Yaskawa INFORM job: A_ROOF_SIDE_0617_2_PAINT_28.JBI

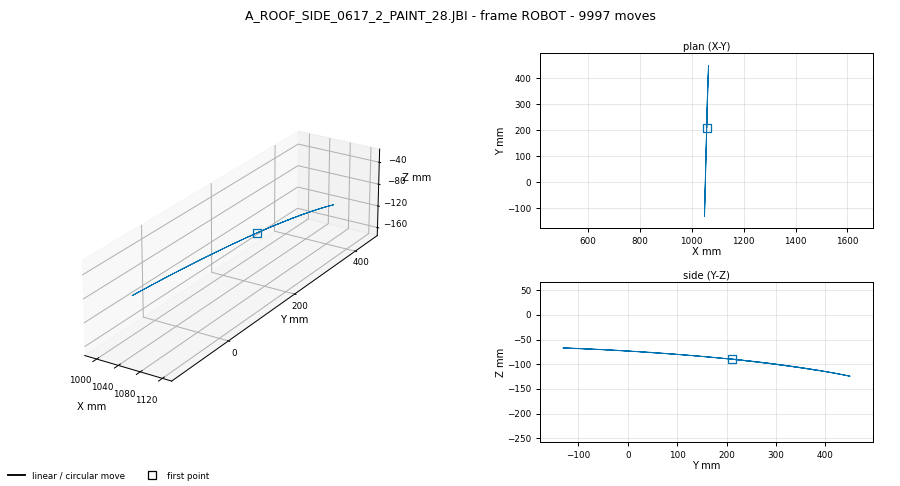
[picture p0: tool path of A_ROOF_SIDE_0617_2_PAINT_28.JBI in frame ROBOT, 9997 of 9997 moves have a stored position in this frame; points joined in program order, loops and branches not executed]
/JOB
//NAME A_ROOF_SIDE_0617_2_PAINT28
//POS
///NPOS 9997,0,0,0,0,0
///TOOL 1
///USER 0
///POSTYPE ROBOT
///RECTAN
///RCONF 1,0,0,0,0,0,0,0,0,0,0,0,0,0,0,0,0,0,0,0,0,0,0,0
C00000=1058.652,210.602,-89.176,172.510,33.165,156.166
C00001=1058.658,210.851,-89.202,172.512,33.168,156.167
C00002=1058.665,211.100,-89.228,172.514,33.173,156.168
C00003=1058.671,211.349,-89.254,172.516,33.176,156.168
C00004=1058.677,211.597,-89.280,172.518,33.181,156.169
C00005=1058.683,211.846,-89.306,172.520,33.184,156.170
C00006=1058.690,212.094,-89.332,172.522,33.189,156.171
C00007=1058.695,212.343,-89.358,172.524,33.192,156.171
C00008=1058.702,212.591,-89.384,172.526,33.196,156.172
C00009=1058.708,212.840,-89.410,172.528,33.200,156.173
C00010=1058.714,213.088,-89.436,172.530,33.204,156.174
C00011=1058.721,213.337,-89.461,172.531,33.208,156.174
C00012=1058.726,213.585,-89.488,172.533,33.212,156.175
C00013=1058.733,213.834,-89.513,172.535,33.216,156.176
C00014=1058.738,214.082,-89.540,172.537,33.220,156.177
C00015=1058.745,214.331,-89.565,172.539,33.224,156.177
C00016=1058.751,214.580,-89.592,172.541,33.227,156.178
C00017=1058.759,214.908,-89.627,172.544,33.233,156.179
C00018=1058.767,215.238,-89.662,172.546,33.238,156.180
C00019=1058.775,215.566,-89.696,172.549,33.243,156.181
C00020=1058.783,215.895,-89.731,172.553,33.248,156.182
C00021=1058.789,216.144,-89.756,172.555,33.253,156.183
C00022=1058.795,216.392,-89.783,172.557,33.256,156.184
C00023=1058.802,216.641,-89.810,172.559,33.260,156.184
C00024=1058.808,216.890,-89.835,172.561,33.264,156.185
C00025=1058.814,217.138,-89.862,172.563,33.268,156.186
C00026=1058.820,217.386,-89.888,172.565,33.271,156.186
C00027=1058.827,217.636,-89.914,172.567,33.276,156.187
C00028=1058.832,217.884,-89.941,172.569,33.279,156.188
C00029=1058.839,218.132,-89.967,172.571,33.284,156.189
C00030=1058.845,218.380,-89.993,172.573,33.287,156.189
C00031=1058.851,218.630,-90.019,172.575,33.291,156.190
C00032=1058.857,218.878,-90.046,172.577,33.295,156.191
C00033=1058.864,219.126,-90.072,172.579,33.299,156.192
C00034=1058.870,219.375,-90.099,172.581,33.302,156.192
C00035=1058.876,219.624,-90.125,172.583,33.307,156.193
C00036=1058.882,219.872,-90.151,172.585,33.310,156.194
C00037=1058.888,220.121,-90.177,172.587,33.314,156.194
C00038=1058.895,220.369,-90.204,172.589,33.318,156.195
C00039=1058.901,220.618,-90.230,172.591,33.322,156.196
C00040=1058.907,220.866,-90.256,172.593,33.326,156.197
C00041=1058.914,221.102,-90.282,172.595,33.329,156.197
C00042=1058.918,221.337,-90.307,172.598,33.333,156.198
C00043=1058.925,221.573,-90.333,172.600,33.337,156.199
C00044=1058.930,221.809,-90.357,172.601,33.340,156.199
C00045=1058.936,222.045,-90.382,172.603,33.344,156.200
C00046=1058.942,222.280,-90.407,172.605,33.348,156.201
C00047=1058.948,222.516,-90.433,172.607,33.351,156.202
C00048=1058.954,222.752,-90.458,172.609,33.355,156.202
C00049=1058.959,223.000,-90.485,172.611,33.359,156.203
C00050=1058.966,223.249,-90.512,172.613,33.363,156.204
C00051=1058.972,223.498,-90.538,172.615,33.367,156.205
C00052=1058.977,223.746,-90.565,172.617,33.371,156.205
C00053=1058.985,223.995,-90.591,172.619,33.374,156.206
C00054=1058.990,224.243,-90.618,172.621,33.379,156.207
C00055=1058.996,224.491,-90.645,172.623,33.382,156.207
C00056=1059.003,224.740,-90.672,172.626,33.386,156.208
C00057=1059.009,224.988,-90.699,172.628,33.390,156.209
C00058=1059.016,225.237,-90.725,172.630,33.394,156.210
C00059=1059.021,225.485,-90.752,172.632,33.397,156.210
C00060=1059.027,225.734,-90.779,172.635,33.402,156.211
C00061=1059.034,225.983,-90.806,172.637,33.405,156.212
C00062=1059.039,226.231,-90.832,172.639,33.409,156.212
C00063=1059.045,226.479,-90.859,172.641,33.413,156.213
C00064=1059.053,226.728,-90.886,172.643,33.417,156.214
C00065=1059.058,226.976,-90.913,172.645,33.421,156.215
C00066=1059.065,227.225,-90.940,172.647,33.424,156.215
C00067=1059.070,227.473,-90.966,172.649,33.428,156.216
C00068=1059.077,227.722,-90.993,172.651,33.432,156.217
C00069=1059.083,227.970,-91.021,172.654,33.436,156.218
C00070=1059.090,228.219,-91.047,172.656,33.439,156.218
C00071=1059.096,228.467,-91.074,172.658,33.444,156.219
C00072=1059.102,228.716,-91.101,172.660,33.447,156.220
C00073=1059.108,228.964,-91.128,172.662,33.451,156.220
C00074=1059.114,229.212,-91.155,172.664,33.455,156.221
C00075=1059.120,229.461,-91.182,172.666,33.459,156.222
C00076=1059.126,229.710,-91.209,172.669,33.463,156.223
C00077=1059.133,229.958,-91.236,172.671,33.466,156.223
C00078=1059.139,230.207,-91.263,172.673,33.470,156.224
C00079=1059.145,230.456,-91.290,172.676,33.474,156.225
C00080=1059.151,230.703,-91.317,172.678,33.478,156.226
C00081=1059.157,230.952,-91.344,172.680,33.482,156.226
C00082=1059.164,231.200,-91.372,172.682,33.486,156.227
C00083=1059.170,231.449,-91.399,172.684,33.489,156.228
C00084=1059.176,231.698,-91.425,172.686,33.494,156.229
C00085=1059.182,231.946,-91.453,172.688,33.497,156.229
C00086=1059.188,232.194,-91.480,172.690,33.501,156.230
C00087=1059.194,232.443,-91.508,172.693,33.505,156.231
C00088=1059.200,232.692,-91.535,172.695,33.509,156.231
C00089=1059.207,232.940,-91.562,172.697,33.512,156.232
C00090=1059.212,233.188,-91.589,172.700,33.516,156.233
C00091=1059.219,233.437,-91.617,172.702,33.520,156.234
C00092=1059.225,233.685,-91.643,172.704,33.524,156.234
C00093=1059.231,233.934,-91.671,172.706,33.528,156.235
C00094=1059.236,234.182,-91.698,172.708,33.532,156.236
C00095=1059.243,234.431,-91.726,172.711,33.536,156.237
C00096=1059.249,234.679,-91.753,172.713,33.539,156.237
C00097=1059.255,234.911,-91.779,172.715,33.543,156.238
C00098=1059.261,235.142,-91.804,172.717,33.546,156.239
C00099=1059.266,235.375,-91.830,172.719,33.550,156.239
C00100=1059.272,235.606,-91.856,172.721,33.554,156.240
C00101=1059.278,235.838,-91.881,172.723,33.557,156.241
C00102=1059.284,236.070,-91.907,172.725,33.560,156.241
C00103=1059.290,236.301,-91.932,172.728,33.564,156.242
C00104=1059.295,236.532,-91.958,172.730,33.568,156.243
C00105=1059.301,236.782,-91.985,172.732,33.571,156.243
C00106=1059.307,237.030,-92.013,172.734,33.576,156.244
C00107=1059.314,237.278,-92.041,172.736,33.579,156.245
C00108=1059.320,237.527,-92.068,172.739,33.583,156.246
C00109=1059.325,237.775,-92.096,172.741,33.587,156.246
C00110=1059.332,238.023,-92.123,172.743,33.591,156.247
C00111=1059.339,238.272,-92.151,172.745,33.594,156.248
C00112=1059.344,238.520,-92.178,172.747,33.598,156.248
C00113=1059.350,238.769,-92.206,172.750,33.602,156.249
C00114=1059.357,239.017,-92.234,172.752,33.606,156.250
C00115=1059.363,239.265,-92.261,172.755,33.610,156.251
C00116=1059.370,239.514,-92.289,172.757,33.613,156.251
C00117=1059.375,239.763,-92.316,172.759,33.617,156.252
C00118=1059.382,240.011,-92.344,172.762,33.621,156.253
C00119=1059.388,240.259,-92.372,172.764,33.625,156.254
C00120=1059.394,240.508,-92.400,172.766,33.628,156.254
C00121=1059.400,240.756,-92.427,172.768,33.632,156.255
C00122=1059.407,241.004,-92.455,172.770,33.636,156.256
C00123=1059.413,241.253,-92.483,172.773,33.640,156.256
C00124=1059.419,241.501,-92.510,172.775,33.644,156.257
C00125=1059.425,241.750,-92.538,172.777,33.647,156.258
C00126=1059.431,241.998,-92.566,172.780,33.651,156.259
C00127=1059.437,242.246,-92.593,172.783,33.655,156.259
C00128=1059.443,242.495,-92.622,172.785,33.659,156.260
C00129=1059.450,242.743,-92.649,172.787,33.662,156.261
C00130=1059.455,242.991,-92.677,172.789,33.666,156.261
C00131=1059.462,243.240,-92.705,172.791,33.670,156.262
C00132=1059.468,243.489,-92.733,172.794,33.674,156.263
C00133=1059.475,243.737,-92.761,172.796,33.678,156.264
C00134=1059.480,243.985,-92.789,172.798,33.682,156.265
C00135=1059.487,244.234,-92.817,172.800,33.685,156.265
C00136=1059.493,244.482,-92.845,172.803,33.689,156.266
C00137=1059.498,244.730,-92.874,172.806,33.693,156.267
C00138=1059.505,244.978,-92.902,172.808,33.697,156.267
C00139=1059.511,245.227,-92.930,172.810,33.701,156.268
C00140=1059.517,245.475,-92.958,172.813,33.704,156.269
C00141=1059.523,245.723,-92.986,172.815,33.708,156.270
C00142=1059.530,245.972,-93.013,172.817,33.712,156.270
C00143=1059.535,246.221,-93.042,172.819,33.716,156.271
C00144=1059.542,246.469,-93.071,172.822,33.719,156.272
C00145=1059.547,246.717,-93.099,172.824,33.724,156.273
C00146=1059.554,246.965,-93.126,172.826,33.727,156.273
C00147=1059.560,247.214,-93.155,172.829,33.731,156.274
C00148=1059.566,247.463,-93.183,172.832,33.735,156.275
C00149=1059.571,247.710,-93.212,172.834,33.739,156.275
C00150=1059.578,247.959,-93.239,172.836,33.743,156.276
C00151=1059.584,248.207,-93.268,172.839,33.747,156.277
C00152=1059.590,248.456,-93.297,172.841,33.750,156.278
C00153=1059.595,248.684,-93.323,172.843,33.754,156.278
C00154=1059.601,248.913,-93.348,172.845,33.757,156.279
C00155=1059.607,249.142,-93.375,172.847,33.761,156.280
C00156=1059.611,249.370,-93.401,172.850,33.765,156.280
C00157=1059.618,249.599,-93.427,172.852,33.768,156.281
C00158=1059.623,249.828,-93.453,172.854,33.771,156.282
C00159=1059.629,250.057,-93.479,172.857,33.775,156.282
C00160=1059.634,250.285,-93.505,172.859,33.779,156.283
C00161=1059.640,250.534,-93.534,172.861,33.782,156.284
C00162=1059.647,250.782,-93.563,172.863,33.786,156.285
C00163=1059.653,251.030,-93.591,172.866,33.790,156.285
C00164=1059.659,251.278,-93.620,172.868,33.794,156.286
C00165=1059.665,251.526,-93.647,172.870,33.797,156.287
C00166=1059.671,251.774,-93.677,172.873,33.802,156.288
C00167=1059.677,252.023,-93.705,172.876,33.805,156.288
C00168=1059.683,252.271,-93.734,172.878,33.809,156.289
C00169=1059.689,252.520,-93.762,172.880,33.812,156.290
C00170=1059.695,252.768,-93.791,172.883,33.817,156.291
C00171=1059.702,253.017,-93.819,172.885,33.820,156.291
C00172=1059.708,253.265,-93.848,172.887,33.824,156.292
C00173=1059.714,253.513,-93.876,172.890,33.828,156.293
C00174=1059.720,253.761,-93.905,172.893,33.832,156.293
C00175=1059.726,254.009,-93.934,172.895,33.835,156.294
C00176=1059.732,254.258,-93.962,172.898,33.839,156.295
C00177=1059.738,254.506,-93.991,172.900,33.843,156.296
C00178=1059.745,254.754,-94.019,172.903,33.847,156.296
C00179=1059.751,255.003,-94.048,172.905,33.851,156.297
C00180=1059.758,255.251,-94.077,172.907,33.854,156.298
C00181=1059.764,255.499,-94.106,172.910,33.858,156.299
C00182=1059.770,255.748,-94.135,172.912,33.862,156.299
C00183=1059.776,255.996,-94.164,172.915,33.866,156.300
C00184=1059.782,256.244,-94.192,172.918,33.869,156.301
C00185=1059.788,256.493,-94.221,172.920,33.874,156.302
C00186=1059.794,256.741,-94.250,172.922,33.877,156.302
C00187=1059.801,256.989,-94.279,172.925,33.881,156.303
C00188=1059.807,257.237,-94.307,172.927,33.884,156.304
C00189=1059.814,257.485,-94.336,172.930,33.888,156.304
C00190=1059.820,257.734,-94.365,172.932,33.892,156.305
C00191=1059.826,257.982,-94.394,172.935,33.896,156.306
C00192=1059.832,258.230,-94.422,172.938,33.900,156.307
C00193=1059.838,258.479,-94.451,172.940,33.903,156.307
C00194=1059.845,258.727,-94.480,172.943,33.907,156.308
C00195=1059.851,258.975,-94.509,172.945,33.911,156.309
C00196=1059.857,259.223,-94.538,172.947,33.915,156.309
C00197=1059.863,259.471,-94.567,172.950,33.918,156.310
C00198=1059.869,259.720,-94.596,172.952,33.922,156.311
C00199=1059.876,259.968,-94.625,172.956,33.926,156.312
C00200=1059.883,260.216,-94.653,172.958,33.930,156.312
C00201=1059.889,260.465,-94.683,172.961,33.933,156.313
C00202=1059.896,260.713,-94.712,172.963,33.937,156.314
C00203=1059.902,260.961,-94.741,172.965,33.941,156.315
C00204=1059.908,261.209,-94.770,172.968,33.944,156.315
C00205=1059.914,261.457,-94.799,172.970,33.948,156.316
C00206=1059.921,261.705,-94.828,172.973,33.952,156.317
C00207=1059.927,261.953,-94.857,172.976,33.956,156.317
C00208=1059.933,262.202,-94.886,172.979,33.959,156.318
C00209=1059.939,262.430,-94.913,172.981,33.963,156.319
C00210=1059.945,262.657,-94.940,172.983,33.966,156.319
C00211=1059.951,262.885,-94.966,172.985,33.970,156.320
C00212=1059.957,263.113,-94.993,172.988,33.973,156.321
C00213=1059.963,263.340,-95.019,172.990,33.976,156.321
C00214=1059.968,263.568,-95.046,172.992,33.980,156.322
C00215=1059.974,263.796,-95.073,172.995,33.983,156.323
C00216=1059.979,264.023,-95.101,172.998,33.987,156.324
C00217=1059.985,264.271,-95.130,173.000,33.991,156.324
C00218=1059.992,264.519,-95.159,173.002,33.995,156.325
C00219=1059.998,264.768,-95.188,173.005,33.999,156.326
C00220=1060.003,265.016,-95.218,173.007,34.002,156.326
C00221=1060.010,265.265,-95.247,173.010,34.006,156.327
C00222=1060.017,265.512,-95.277,173.013,34.010,156.328
C00223=1060.022,265.761,-95.307,173.016,34.014,156.329
C00224=1060.029,266.009,-95.336,173.018,34.017,156.329
C00225=1060.035,266.257,-95.365,173.021,34.021,156.330
C00226=1060.041,266.505,-95.395,173.023,34.025,156.331
C00227=1060.048,266.754,-95.424,173.026,34.029,156.332
C00228=1060.054,267.002,-95.453,173.028,34.033,156.332
C00229=1060.060,267.250,-95.484,173.032,34.036,156.333
C00230=1060.066,267.498,-95.513,173.034,34.040,156.334
C00231=1060.072,267.746,-95.542,173.037,34.044,156.335
C00232=1060.079,267.994,-95.572,173.039,34.048,156.335
C00233=1060.085,268.243,-95.602,173.042,34.052,156.336
C00234=1060.091,268.491,-95.631,173.044,34.055,156.337
C00235=1060.097,268.739,-95.661,173.047,34.059,156.338
C00236=1060.103,268.987,-95.690,173.050,34.063,156.338
C00237=1060.110,269.235,-95.720,173.053,34.067,156.339
C00238=1060.116,269.483,-95.750,173.055,34.071,156.340
C00239=1060.122,269.731,-95.780,173.058,34.074,156.341
C00240=1060.128,269.979,-95.809,173.060,34.079,156.341
C00241=1060.135,270.227,-95.839,173.063,34.082,156.342
C00242=1060.141,270.476,-95.869,173.065,34.086,156.343
C00243=1060.147,270.723,-95.899,173.069,34.090,156.344
C00244=1060.153,270.972,-95.928,173.071,34.094,156.344
C00245=1060.160,271.220,-95.958,173.074,34.097,156.345
C00246=1060.165,271.469,-95.988,173.076,34.101,156.346
C00247=1060.172,271.716,-96.018,173.079,34.105,156.347
C00248=1060.178,271.965,-96.048,173.081,34.109,156.347
C00249=1060.184,272.213,-96.078,173.085,34.113,156.348
C00250=1060.190,272.461,-96.108,173.087,34.116,156.349
C00251=1060.197,272.709,-96.137,173.090,34.120,156.350
C00252=1060.203,272.957,-96.168,173.092,34.124,156.350
C00253=1060.210,273.205,-96.198,173.095,34.128,156.351
C00254=1060.215,273.453,-96.227,173.097,34.132,156.352
C00255=1060.221,273.702,-96.258,173.101,34.136,156.353
C00256=1060.228,273.949,-96.288,173.104,34.139,156.353
C00257=1060.234,274.198,-96.317,173.106,34.143,156.354
C00258=1060.240,274.446,-96.348,173.109,34.147,156.355
C00259=1060.247,274.694,-96.378,173.111,34.151,156.356
C00260=1060.252,274.941,-96.408,173.114,34.155,156.356
C00261=1060.258,275.191,-96.438,173.116,34.158,156.357
C00262=1060.265,275.438,-96.468,173.120,34.163,156.358
C00263=1060.271,275.686,-96.498,173.123,34.166,156.359
C00264=1060.277,275.934,-96.529,173.125,34.170,156.360
C00265=1060.284,276.164,-96.557,173.127,34.174,156.360
C00266=1060.289,276.394,-96.584,173.130,34.178,156.361
C00267=1060.295,276.623,-96.612,173.132,34.181,156.362
C00268=1060.300,276.852,-96.640,173.136,34.184,156.362
C00269=1060.306,277.082,-96.669,173.138,34.188,156.363
C00270=1060.311,277.312,-96.696,173.140,34.191,156.364
C00271=1060.317,277.541,-96.724,173.143,34.195,156.364
C00272=1060.323,277.771,-96.753,173.145,34.199,156.365
C00273=1060.330,278.019,-96.783,173.148,34.203,156.366
C00274=1060.336,278.266,-96.813,173.151,34.206,156.367
C00275=1060.342,278.515,-96.844,173.154,34.211,156.367
C00276=1060.348,278.763,-96.874,173.157,34.214,156.368
C00277=1060.355,279.011,-96.904,173.159,34.218,156.369
C00278=1060.361,279.259,-96.935,173.162,34.222,156.370
C00279=1060.367,279.507,-96.965,173.165,34.226,156.370
C00280=1060.373,279.755,-96.996,173.168,34.230,156.371
C00281=1060.380,280.003,-97.026,173.171,34.233,156.372
C00282=1060.386,280.251,-97.056,173.173,34.237,156.373
C00283=1060.392,280.499,-97.086,173.176,34.241,156.374
C00284=1060.398,280.748,-97.117,173.179,34.245,156.374
C00285=1060.404,280.995,-97.147,173.181,34.249,156.375
C00286=1060.411,281.243,-97.179,173.185,34.253,156.376
C00287=1060.417,281.491,-97.209,173.187,34.257,156.377
C00288=1060.423,281.740,-97.240,173.190,34.261,156.377
C00289=1060.429,281.987,-97.270,173.193,34.264,156.378
C00290=1060.435,282.236,-97.301,173.195,34.269,156.379
C00291=1060.442,282.483,-97.332,173.199,34.272,156.380
C00292=1060.448,282.732,-97.363,173.202,34.276,156.381
C00293=1060.454,282.979,-97.393,173.204,34.280,156.381
C00294=1060.460,283.228,-97.424,173.207,34.284,156.382
C00295=1060.466,283.475,-97.455,173.210,34.288,156.383
C00296=1060.473,283.724,-97.486,173.213,34.292,156.384
C00297=1060.479,283.972,-97.516,173.216,34.296,156.384
C00298=1060.485,284.219,-97.547,173.219,34.300,156.385
C00299=1060.491,284.467,-97.578,173.221,34.304,156.386
C00300=1060.498,284.716,-97.609,173.224,34.307,156.387
C00301=1060.504,284.963,-97.640,173.227,34.312,156.388
C00302=1060.510,285.212,-97.670,173.230,34.315,156.388
C00303=1060.517,285.459,-97.702,173.233,34.319,156.389
C00304=1060.523,285.707,-97.732,173.236,34.323,156.390
C00305=1060.529,285.956,-97.763,173.238,34.327,156.391
C00306=1060.535,286.203,-97.794,173.241,34.331,156.391
C00307=1060.542,286.451,-97.825,173.245,34.335,156.392
C00308=1060.548,286.699,-97.856,173.247,34.338,156.393
C00309=1060.554,286.947,-97.886,173.250,34.343,156.394
C00310=1060.561,287.195,-97.918,173.253,34.347,156.395
C00311=1060.567,287.444,-97.949,173.256,34.350,156.395
C00312=1060.573,287.691,-97.980,173.259,34.355,156.396
C00313=1060.580,287.939,-98.010,173.262,34.358,156.397
C00314=1060.587,288.187,-98.042,173.265,34.362,156.398
C00315=1060.592,288.435,-98.073,173.267,34.366,156.398
C00316=1060.598,288.683,-98.104,173.270,34.370,156.399
C00317=1060.604,288.930,-98.135,173.274,34.374,156.400
C00318=1060.611,289.179,-98.166,173.277,34.378,156.401
C00319=1060.618,289.427,-98.197,173.279,34.382,156.402
C00320=1060.623,289.674,-98.229,173.282,34.386,156.402
C00321=1060.629,289.910,-98.258,173.285,34.390,156.403
C00322=1060.636,290.145,-98.288,173.288,34.393,156.404
C00323=1060.641,290.380,-98.317,173.291,34.397,156.405
C00324=1060.647,290.615,-98.347,173.293,34.401,156.405
C00325=1060.653,290.850,-98.377,173.296,34.405,156.406
C00326=1060.659,291.084,-98.406,173.299,34.408,156.407
C00327=1060.665,291.320,-98.437,173.302,34.412,156.408
C00328=1060.671,291.555,-98.466,173.305,34.416,156.408
C00329=1060.677,291.802,-98.497,173.308,34.420,156.409
C00330=1060.683,292.050,-98.529,173.310,34.424,156.410
C00331=1060.690,292.298,-98.560,173.313,34.428,156.411
C00332=1060.697,292.546,-98.592,173.317,34.432,156.412
C00333=1060.702,292.794,-98.623,173.320,34.436,156.412
C00334=1060.709,293.042,-98.655,173.322,34.440,156.413
C00335=1060.715,293.290,-98.685,173.325,34.444,156.414
C00336=1060.721,293.538,-98.717,173.328,34.447,156.415
C00337=1060.727,293.786,-98.748,173.332,34.452,156.416
C00338=1060.734,294.033,-98.780,173.335,34.456,156.416
C00339=1060.740,294.282,-98.812,173.337,34.459,156.417
C00340=1060.747,294.530,-98.843,173.340,34.463,156.418
C00341=1060.753,294.777,-98.874,173.344,34.468,156.419
C00342=1060.759,295.025,-98.906,173.347,34.472,156.420
C00343=1060.765,295.273,-98.938,173.350,34.475,156.420
C00344=1060.771,295.521,-98.970,173.352,34.479,156.421
C00345=1060.778,295.769,-99.001,173.355,34.484,156.422
C00346=1060.784,296.017,-99.033,173.359,34.488,156.423
C00347=1060.790,296.264,-99.064,173.362,34.491,156.424
C00348=1060.796,296.513,-99.096,173.365,34.495,156.425
C00349=1060.803,296.760,-99.129,173.367,34.500,156.425
C00350=1060.809,297.008,-99.161,173.371,34.504,156.426
C00351=1060.815,297.255,-99.192,173.374,34.508,156.427
C00352=1060.821,297.504,-99.224,173.377,34.512,156.428
C00353=1060.827,297.752,-99.256,173.380,34.516,156.429
C00354=1060.834,297.999,-99.288,173.382,34.520,156.429
C00355=1060.840,298.247,-99.320,173.386,34.524,156.430
C00356=1060.846,298.495,-99.352,173.389,34.528,156.431
C00357=1060.852,298.743,-99.384,173.392,34.532,156.432
C00358=1060.859,298.990,-99.416,173.395,34.536,156.433
C00359=1060.865,299.238,-99.448,173.399,34.540,156.434
C00360=1060.871,299.487,-99.480,173.401,34.545,156.435
C00361=1060.877,299.734,-99.513,173.404,34.549,156.435
C00362=1060.883,299.981,-99.544,173.407,34.553,156.436
C00363=1060.889,300.230,-99.576,173.411,34.557,156.437
C00364=1060.895,300.477,-99.608,173.414,34.561,156.438
C00365=1060.901,300.725,-99.640,173.417,34.565,156.439
C00366=1060.908,300.973,-99.673,173.419,34.569,156.440
C00367=1060.915,301.221,-99.705,173.423,34.574,156.440
C00368=1060.920,301.469,-99.737,173.426,34.578,156.441
C00369=1060.927,301.717,-99.769,173.429,34.582,156.442
C00370=1060.932,301.964,-99.801,173.432,34.586,156.443
C00371=1060.938,302.212,-99.834,173.436,34.590,156.444
C00372=1060.945,302.460,-99.865,173.439,34.594,156.445
C00373=1060.951,302.707,-99.898,173.441,34.598,156.445
C00374=1060.958,302.955,-99.931,173.444,34.602,156.446
C00375=1060.964,303.203,-99.963,173.448,34.607,156.447
C00376=1060.970,303.451,-99.995,173.451,34.611,156.448
C00377=1060.977,303.693,-100.026,173.454,34.615,156.449
C00378=1060.983,303.936,-100.058,173.457,34.618,156.450
C00379=1060.989,304.178,-100.090,173.460,34.623,156.450
C00380=1060.995,304.421,-100.122,173.464,34.627,156.451
C00381=1061.001,304.664,-100.153,173.466,34.631,156.452
C00382=1061.007,304.906,-100.185,173.469,34.635,156.453
C00383=1061.013,305.149,-100.217,173.473,34.639,156.454
C00384=1061.019,305.392,-100.248,173.476,34.643,156.455
C00385=1061.026,305.639,-100.281,173.479,34.647,156.456
C00386=1061.033,305.887,-100.313,173.482,34.651,156.456
C00387=1061.039,306.135,-100.346,173.486,34.656,156.457
C00388=1061.045,306.383,-100.378,173.489,34.660,156.458
C00389=1061.051,306.630,-100.411,173.492,34.664,156.459
C00390=1061.058,306.878,-100.444,173.495,34.668,156.460
C00391=1061.064,307.126,-100.477,173.499,34.672,156.461
C00392=1061.071,307.374,-100.509,173.502,34.676,156.461
C00393=1061.077,307.622,-100.541,173.504,34.680,156.462
C00394=1061.084,307.869,-100.574,173.507,34.684,156.463
C00395=1061.090,308.117,-100.606,173.511,34.689,156.464
C00396=1061.096,308.364,-100.639,173.514,34.693,156.465
C00397=1061.103,308.612,-100.672,173.517,34.697,156.466
C00398=1061.109,308.860,-100.705,173.520,34.701,156.467
C00399=1061.116,309.108,-100.738,173.524,34.705,156.467
C00400=1061.123,309.355,-100.770,173.527,34.709,156.468
C00401=1061.129,309.603,-100.803,173.530,34.713,156.469
C00402=1061.135,309.850,-100.835,173.533,34.717,156.470
C00403=1061.141,310.099,-100.867,173.537,34.722,156.471
C00404=1061.148,310.347,-100.900,173.540,34.726,156.472
C00405=1061.155,310.595,-100.933,173.543,34.730,156.473
C00406=1061.161,310.842,-100.967,173.547,34.734,156.473
C00407=1061.167,311.089,-100.999,173.550,34.739,156.474
C00408=1061.174,311.337,-101.032,173.553,34.743,156.475
C00409=1061.181,311.585,-101.065,173.556,34.747,156.476
C00410=1061.187,311.833,-101.098,173.560,34.751,156.477
C00411=1061.193,312.080,-101.131,173.563,34.755,156.478
C00412=1061.200,312.328,-101.164,173.566,34.759,156.479
C00413=1061.207,312.576,-101.196,173.570,34.764,156.480
C00414=1061.213,312.823,-101.229,173.573,34.768,156.480
C00415=1061.220,313.072,-101.262,173.576,34.772,156.481
C00416=1061.227,313.319,-101.295,173.580,34.776,156.482
C00417=1061.233,313.566,-101.328,173.584,34.780,156.483
C00418=1061.240,313.815,-101.361,173.587,34.784,156.484
C00419=1061.246,314.062,-101.394,173.590,34.789,156.485
C00420=1061.252,314.309,-101.428,173.593,34.793,156.486
C00421=1061.258,314.557,-101.461,173.597,34.798,156.487
C00422=1061.265,314.806,-101.494,173.600,34.802,156.487
C00423=1061.271,315.053,-101.528,173.603,34.807,156.488
C00424=1061.277,315.300,-101.561,173.607,34.811,156.489
C00425=1061.283,315.548,-101.594,173.610,34.815,156.490
C00426=1061.290,315.796,-101.628,173.613,34.820,156.491
C00427=1061.296,316.044,-101.661,173.617,34.824,156.492
C00428=1061.302,316.291,-101.695,173.620,34.828,156.493
C00429=1061.309,316.539,-101.728,173.623,34.832,156.494
C00430=1061.315,316.786,-101.762,173.627,34.837,156.495
C00431=1061.321,317.034,-101.795,173.630,34.841,156.496
C00432=1061.327,317.282,-101.829,173.633,34.846,156.497
C00433=1061.333,317.526,-101.862,173.636,34.850,156.497
C00434=1061.340,317.771,-101.895,173.640,34.855,156.498
C00435=1061.345,318.015,-101.928,173.643,34.859,156.499
C00436=1061.352,318.260,-101.961,173.646,34.863,156.500
C00437=1061.359,318.504,-101.995,173.650,34.867,156.501
C00438=1061.365,318.749,-102.027,173.653,34.872,156.502
C00439=1061.371,318.994,-102.061,173.656,34.876,156.503
C00440=1061.377,319.238,-102.094,173.660,34.880,156.504
C00441=1061.383,319.485,-102.128,173.663,34.885,156.505
C00442=1061.390,319.733,-102.162,173.666,34.889,156.506
C00443=1061.396,319.981,-102.195,173.671,34.894,156.507
C00444=1061.403,320.229,-102.229,173.674,34.898,156.508
C00445=1061.409,320.476,-102.263,173.677,34.902,156.508
C00446=1061.416,320.724,-102.297,173.681,34.907,156.509
C00447=1061.422,320.972,-102.330,173.684,34.911,156.510
C00448=1061.429,321.219,-102.364,173.687,34.916,156.511
C00449=1061.435,321.466,-102.398,173.691,34.921,156.512
C00450=1061.442,321.714,-102.432,173.694,34.925,156.513
C00451=1061.447,321.962,-102.465,173.697,34.929,156.514
C00452=1061.454,322.210,-102.499,173.701,34.933,156.515
C00453=1061.460,322.457,-102.533,173.705,34.938,156.516
C00454=1061.467,322.705,-102.567,173.708,34.943,156.517
C00455=1061.474,322.952,-102.601,173.711,34.947,156.518
C00456=1061.480,323.200,-102.635,173.715,34.951,156.519
C00457=1061.487,323.447,-102.669,173.718,34.956,156.520
C00458=1061.493,323.695,-102.703,173.721,34.960,156.521
C00459=1061.499,323.944,-102.737,173.726,34.965,156.522
C00460=1061.506,324.191,-102.770,173.729,34.969,156.523
C00461=1061.512,324.439,-102.805,173.732,34.974,156.523
C00462=1061.519,324.685,-102.838,173.736,34.978,156.524
C00463=1061.525,324.933,-102.873,173.739,34.983,156.525
C00464=1061.532,325.181,-102.907,173.742,34.987,156.526
C00465=1061.538,325.428,-102.940,173.747,34.992,156.527
C00466=1061.545,325.676,-102.976,173.750,34.996,156.528
C00467=1061.552,325.923,-103.009,173.754,35.001,156.529
C00468=1061.558,326.171,-103.043,173.757,35.005,156.530
C00469=1061.565,326.419,-103.078,173.760,35.010,156.531
C00470=1061.572,326.666,-103.112,173.765,35.014,156.532
C00471=1061.578,326.914,-103.146,173.768,35.019,156.533
C00472=1061.585,327.161,-103.180,173.771,35.023,156.534
C00473=1061.591,327.409,-103.214,173.775,35.028,156.535
C00474=1061.598,327.657,-103.249,173.779,35.032,156.536
C00475=1061.605,327.904,-103.283,173.782,35.037,156.537
C00476=1061.611,328.152,-103.317,173.786,35.041,156.538
C00477=1061.618,328.400,-103.351,173.789,35.046,156.539
C00478=1061.625,328.647,-103.386,173.792,35.050,156.540
C00479=1061.631,328.894,-103.420,173.797,35.055,156.541
C00480=1061.638,329.142,-103.454,173.800,35.059,156.542
C00481=1061.645,329.390,-103.488,173.803,35.064,156.543
C00482=1061.651,329.637,-103.523,173.807,35.068,156.544
C00483=1061.658,329.885,-103.558,173.811,35.073,156.545
C00484=1061.665,330.132,-103.591,173.815,35.077,156.546
C00485=1061.671,330.379,-103.626,173.818,35.082,156.547
C00486=1061.678,330.627,-103.661,173.822,35.087,156.547
C00487=1061.685,330.875,-103.696,173.826,35.091,156.548
C00488=1061.691,331.123,-103.730,173.829,35.096,156.549
C00489=1061.697,331.364,-103.765,173.832,35.101,156.550
C00490=1061.704,331.606,-103.798,173.836,35.105,156.551
C00491=1061.710,331.847,-103.832,173.840,35.110,156.552
C00492=1061.716,332.089,-103.866,173.844,35.114,156.553
C00493=1061.723,332.331,-103.900,173.847,35.119,156.554
C00494=1061.729,332.572,-103.934,173.850,35.124,156.555
C00495=1061.735,332.814,-103.967,173.854,35.128,156.556
C00496=1061.742,333.056,-104.002,173.858,35.133,156.557
C00497=1061.749,333.303,-104.037,173.861,35.138,156.558
C00498=1061.755,333.550,-104.071,173.865,35.142,156.559
C00499=1061.762,333.798,-104.106,173.869,35.147,156.560
C00500=1061.768,334.045,-104.141,173.873,35.151,156.561
C00501=1061.775,334.293,-104.176,173.876,35.157,156.562
C00502=1061.781,334.541,-104.211,173.879,35.161,156.563
C00503=1061.788,334.788,-104.247,173.884,35.166,156.564
C00504=1061.794,335.035,-104.282,173.887,35.170,156.565
C00505=1061.801,335.283,-104.316,173.891,35.175,156.566
C00506=1061.808,335.531,-104.351,173.895,35.180,156.568
C00507=1061.814,335.778,-104.386,173.898,35.185,156.569
C00508=1061.821,336.026,-104.422,173.902,35.189,156.570
C00509=1061.828,336.273,-104.457,173.906,35.195,156.571
C00510=1061.834,336.520,-104.491,173.910,35.199,156.572
C00511=1061.841,336.767,-104.527,173.913,35.204,156.573
C00512=1061.848,337.014,-104.562,173.917,35.208,156.574
C00513=1061.853,337.263,-104.597,173.921,35.214,156.575
C00514=1061.860,337.510,-104.632,173.925,35.218,156.576
C00515=1061.867,337.757,-104.667,173.929,35.223,156.577
C00516=1061.873,338.004,-104.703,173.932,35.228,156.578
C00517=1061.880,338.252,-104.739,173.937,35.233,156.579
C00518=1061.887,338.499,-104.774,173.940,35.238,156.580
C00519=1061.893,338.747,-104.809,173.943,35.243,156.581
C00520=1061.900,338.994,-104.845,173.948,35.248,156.582
C00521=1061.906,339.241,-104.880,173.951,35.253,156.583
C00522=1061.913,339.489,-104.915,173.956,35.257,156.584
C00523=1061.919,339.737,-104.951,173.959,35.262,156.585
C00524=1061.926,339.984,-104.986,173.962,35.267,156.586
C00525=1061.934,340.231,-105.022,173.967,35.272,156.587
C00526=1061.940,340.479,-105.058,173.970,35.277,156.588
C00527=1061.946,340.726,-105.093,173.975,35.282,156.590
C00528=1061.953,340.974,-105.128,173.978,35.287,156.591
C00529=1061.959,341.221,-105.164,173.982,35.292,156.592
C00530=1061.966,341.468,-105.200,173.986,35.297,156.593
C00531=1061.972,341.716,-105.235,173.990,35.301,156.594
C00532=1061.979,341.963,-105.270,173.994,35.307,156.595
C00533=1061.986,342.210,-105.306,173.997,35.312,156.596
C00534=1061.993,342.458,-105.342,174.002,35.316,156.597
C00535=1061.999,342.706,-105.377,174.005,35.322,156.598
C00536=1062.007,342.952,-105.413,174.009,35.327,156.599
C00537=1062.013,343.200,-105.449,174.013,35.331,156.600
C00538=1062.020,343.447,-105.485,174.017,35.336,156.601
C00539=1062.026,343.695,-105.521,174.021,35.342,156.603
C00540=1062.033,343.942,-105.557,174.025,35.347,156.604
C00541=1062.039,344.190,-105.593,174.029,35.352,156.605
C00542=1062.046,344.436,-105.628,174.033,35.357,156.606
C00543=1062.052,344.684,-105.664,174.037,35.362,156.607
C00544=1062.059,344.931,-105.701,174.041,35.367,156.608
C00545=1062.065,345.171,-105.735,174.044,35.372,156.609
C00546=1062.072,345.410,-105.770,174.048,35.377,156.610
C00547=1062.079,345.649,-105.805,174.052,35.382,156.611
C00548=1062.085,345.888,-105.840,174.056,35.387,156.613
C00549=1062.092,346.127,-105.875,174.060,35.391,156.614
C00550=1062.098,346.367,-105.909,174.063,35.396,156.615
C00551=1062.104,346.606,-105.944,174.068,35.402,156.616
C00552=1062.111,346.846,-105.979,174.071,35.407,156.617
C00553=1062.118,347.093,-106.016,174.076,35.412,156.618
C00554=1062.125,347.340,-106.052,174.079,35.417,156.619
C00555=1062.131,347.588,-106.088,174.084,35.422,156.620
C00556=1062.137,347.835,-106.124,174.087,35.427,156.621
C00557=1062.145,348.082,-106.160,174.092,35.432,156.623
C00558=1062.151,348.329,-106.197,174.095,35.437,156.624
C00559=1062.157,348.576,-106.233,174.100,35.443,156.625
C00560=1062.165,348.824,-106.270,174.103,35.448,156.626
C00561=1062.171,349.071,-106.306,174.108,35.453,156.627
C00562=1062.177,349.319,-106.342,174.111,35.458,156.628
C00563=1062.184,349.566,-106.379,174.116,35.464,156.629
C00564=1062.191,349.813,-106.414,174.120,35.469,156.631
C00565=1062.198,350.061,-106.451,174.124,35.474,156.632
C00566=1062.205,350.308,-106.488,174.128,35.479,156.633
C00567=1062.211,350.555,-106.524,174.132,35.484,156.634
C00568=1062.219,350.802,-106.560,174.136,35.490,156.635
C00569=1062.225,351.049,-106.597,174.140,35.495,156.636
C00570=1062.232,351.297,-106.634,174.144,35.500,156.638
C00571=1062.239,351.544,-106.671,174.149,35.505,156.639
C00572=1062.246,351.791,-106.707,174.152,35.511,156.640
C00573=1062.253,352.038,-106.743,174.157,35.516,156.641
C00574=1062.259,352.285,-106.780,174.160,35.522,156.642
C00575=1062.266,352.533,-106.817,174.165,35.527,156.643
C00576=1062.273,352.779,-106.854,174.169,35.532,156.645
C00577=1062.280,353.027,-106.891,174.173,35.538,156.646
C00578=1062.286,353.274,-106.927,174.177,35.543,156.647
C00579=1062.293,353.521,-106.965,174.182,35.548,156.648
C00580=1062.299,353.768,-107.001,174.186,35.554,156.650
C00581=1062.306,354.016,-107.038,174.190,35.559,156.651
C00582=1062.313,354.263,-107.075,174.194,35.565,156.652
C00583=1062.320,354.510,-107.112,174.198,35.570,156.653
C00584=1062.326,354.757,-107.148,174.203,35.576,156.654
C00585=1062.334,355.005,-107.186,174.206,35.581,156.656
C00586=1062.340,355.252,-107.222,174.211,35.586,156.657
C00587=1062.347,355.499,-107.260,174.215,35.592,156.658
C00588=1062.353,355.746,-107.296,174.219,35.597,156.659
C00589=1062.361,355.993,-107.334,174.224,35.603,156.660
C00590=1062.368,356.241,-107.371,174.228,35.608,156.662
C00591=1062.374,356.487,-107.408,174.232,35.613,156.663
C00592=1062.381,356.735,-107.444,174.236,35.619,156.664
C00593=1062.388,356.981,-107.482,174.241,35.625,156.665
C00594=1062.395,357.228,-107.519,174.244,35.630,156.667
C00595=1062.402,357.476,-107.556,174.249,35.635,156.668
C00596=1062.409,357.723,-107.593,174.254,35.641,156.669
C00597=1062.416,357.970,-107.631,174.257,35.647,156.670
C00598=1062.423,358.218,-107.667,174.262,35.652,156.672
C00599=1062.430,358.464,-107.705,174.266,35.657,156.673
C00600=1062.436,358.711,-107.743,174.271,35.663,156.674
C00601=1062.442,358.953,-107.779,174.274,35.669,156.675
C00602=1062.450,359.195,-107.816,174.279,35.674,156.677
C00603=1062.456,359.436,-107.852,174.284,35.680,156.678
C00604=1062.463,359.677,-107.889,174.287,35.685,156.679
C00605=1062.469,359.919,-107.925,174.292,35.691,156.680
C00606=1062.476,360.161,-107.962,174.295,35.696,156.682
C00607=1062.483,360.402,-107.999,174.300,35.702,156.683
C00608=1062.490,360.643,-108.035,174.305,35.708,156.684
C00609=1062.497,360.890,-108.073,174.309,35.713,156.685
C00610=1062.504,361.137,-108.110,174.313,35.719,156.687
C00611=1062.510,361.384,-108.148,174.317,35.725,156.688
C00612=1062.517,361.631,-108.186,174.322,35.730,156.689
C00613=1062.525,361.878,-108.223,174.327,35.736,156.690
C00614=1062.532,362.125,-108.261,174.330,35.741,156.692
C00615=1062.538,362.373,-108.299,174.335,35.748,156.693
C00616=1062.545,362.619,-108.336,174.340,35.753,156.694
C00617=1062.552,362.866,-108.373,174.344,35.759,156.696
C00618=1062.559,363.114,-108.412,174.349,35.764,156.697
C00619=1062.566,363.360,-108.450,174.353,35.771,156.698
C00620=1062.574,363.607,-108.487,174.357,35.776,156.700
C00621=1062.580,363.855,-108.525,174.362,35.782,156.701
C00622=1062.587,364.102,-108.563,174.366,35.788,156.702
C00623=1062.593,364.349,-108.601,174.371,35.794,156.704
C00624=1062.601,364.595,-108.639,174.375,35.800,156.705
C00625=1062.607,364.842,-108.677,174.379,35.805,156.706
C00626=1062.615,365.090,-108.715,174.384,35.812,156.708
C00627=1062.621,365.336,-108.753,174.389,35.817,156.709
C00628=1062.629,365.584,-108.791,174.393,35.823,156.710
C00629=1062.635,365.830,-108.830,174.398,35.829,156.712
C00630=1062.642,366.077,-108.867,174.402,35.835,156.713
C00631=1062.649,366.324,-108.906,174.406,35.841,156.715
C00632=1062.656,366.571,-108.943,174.411,35.847,156.716
C00633=1062.663,366.818,-108.982,174.416,35.853,156.717
C00634=1062.669,367.065,-109.020,174.420,35.859,156.719
C00635=1062.677,367.312,-109.059,174.425,35.865,156.720
C00636=1062.684,367.559,-109.097,174.430,35.871,156.721
C00637=1062.691,367.806,-109.135,174.435,35.877,156.723
C00638=1062.698,368.052,-109.174,174.438,35.883,156.724
C00639=1062.704,368.300,-109.212,174.443,35.889,156.725
C00640=1062.712,368.546,-109.250,174.448,35.895,156.727
C00641=1062.719,368.793,-109.289,174.452,35.901,156.728
C00642=1062.726,369.040,-109.327,174.457,35.907,156.730
C00643=1062.733,369.287,-109.365,174.462,35.913,156.731
C00644=1062.740,369.534,-109.404,174.466,35.919,156.733
C00645=1062.747,369.780,-109.442,174.471,35.926,156.734
C00646=1062.754,370.027,-109.481,174.476,35.932,156.735
C00647=1062.760,370.275,-109.519,174.481,35.938,156.737
C00648=1062.769,370.522,-109.558,174.485,35.944,156.738
C00649=1062.775,370.769,-109.597,174.490,35.950,156.740
C00650=1062.783,371.015,-109.635,174.495,35.956,156.741
C00651=1062.790,371.262,-109.674,174.500,35.962,156.742
C00652=1062.797,371.509,-109.713,174.504,35.969,156.744
C00653=1062.804,371.755,-109.751,174.508,35.975,156.745
C00654=1062.811,372.002,-109.790,174.513,35.981,156.747
C00655=1062.818,372.250,-109.829,174.517,35.987,156.748
C00656=1062.826,372.496,-109.867,174.522,35.993,156.750
C00657=1062.833,372.749,-109.908,174.528,36.000,156.751
C00658=1062.840,373.004,-109.948,174.533,36.006,156.752
C00659=1062.848,373.258,-109.988,174.538,36.012,156.754
C00660=1062.854,373.511,-110.027,174.542,36.019,156.756
C00661=1062.862,373.758,-110.067,174.547,36.025,156.757
C00662=1062.868,374.005,-110.106,174.552,36.032,156.759
C00663=1062.875,374.252,-110.145,174.557,36.038,156.760
C00664=1062.882,374.499,-110.184,174.562,36.045,156.762
C00665=1062.889,374.745,-110.223,174.566,36.051,156.763
C00666=1062.897,374.993,-110.262,174.571,36.057,156.765
C00667=1062.903,375.239,-110.301,174.576,36.064,156.766
C00668=1062.911,375.486,-110.341,174.581,36.070,156.768
C00669=1062.918,375.732,-110.379,174.586,36.077,156.769
C00670=1062.926,375.979,-110.419,174.590,36.083,156.770
C00671=1062.933,376.226,-110.458,174.595,36.090,156.772
C00672=1062.940,376.472,-110.497,174.600,36.096,156.774
C00673=1062.947,376.720,-110.537,174.605,36.102,156.775
C00674=1062.954,376.966,-110.576,174.610,36.109,156.777
C00675=1062.961,377.213,-110.615,174.614,36.116,156.778
C00676=1062.969,377.460,-110.655,174.620,36.122,156.780
C00677=1062.976,377.706,-110.694,174.625,36.128,156.781
C00678=1062.983,377.953,-110.733,174.630,36.135,156.783
C00679=1062.990,378.199,-110.773,174.635,36.142,156.784
C00680=1062.997,378.446,-110.812,174.640,36.148,156.786
C00681=1063.004,378.694,-110.853,174.644,36.155,156.787
C00682=1063.011,378.940,-110.892,174.649,36.162,156.789
C00683=1063.018,379.187,-110.931,174.654,36.168,156.790
C00684=1063.026,379.433,-110.971,174.659,36.175,156.792
C00685=1063.033,379.680,-111.010,174.665,36.181,156.794
C00686=1063.041,379.927,-111.050,174.670,36.188,156.795
C00687=1063.048,380.173,-111.090,174.674,36.195,156.797
C00688=1063.055,380.420,-111.129,174.679,36.201,156.798
C00689=1063.062,380.666,-111.169,174.684,36.208,156.800
C00690=1063.070,380.913,-111.209,174.689,36.215,156.801
C00691=1063.077,381.160,-111.248,174.695,36.222,156.803
C00692=1063.084,381.407,-111.289,174.700,36.228,156.805
C00693=1063.091,381.653,-111.328,174.705,36.235,156.806
C00694=1063.099,381.900,-111.368,174.710,36.242,156.808
C00695=1063.105,382.146,-111.408,174.715,36.249,156.810
C00696=1063.113,382.393,-111.449,174.721,36.256,156.811
C00697=1063.121,382.639,-111.488,174.725,36.262,156.813
C00698=1063.128,382.886,-111.529,174.730,36.270,156.814
C00699=1063.135,383.133,-111.569,174.735,36.276,156.816
C00700=1063.142,383.379,-111.608,174.740,36.283,156.818
C00701=1063.149,383.626,-111.649,174.746,36.290,156.819
C00702=1063.157,383.872,-111.689,174.751,36.297,156.821
C00703=1063.164,384.119,-111.730,174.756,36.304,156.823
C00704=1063.171,384.366,-111.770,174.761,36.311,156.824
C00705=1063.179,384.612,-111.810,174.767,36.318,156.826
C00706=1063.186,384.859,-111.850,174.772,36.325,156.828
C00707=1063.194,385.106,-111.890,174.777,36.332,156.829
C00708=1063.200,385.352,-111.931,174.782,36.339,156.831
C00709=1063.208,385.599,-111.971,174.788,36.346,156.833
C00710=1063.216,385.845,-112.012,174.793,36.353,156.834
C00711=1063.222,386.091,-112.052,174.798,36.360,156.836
C00712=1063.230,386.338,-112.092,174.804,36.367,156.838
C00713=1063.239,386.623,-112.139,174.809,36.376,156.840
C00714=1063.248,386.907,-112.186,174.815,36.384,156.842
C00715=1063.256,387.191,-112.232,174.821,36.392,156.844
C00716=1063.265,387.476,-112.279,174.827,36.400,156.846
C00717=1063.272,387.722,-112.320,174.833,36.407,156.847
C00718=1063.280,387.969,-112.360,174.838,36.414,156.849
C00719=1063.287,388.216,-112.402,174.844,36.421,156.851
C00720=1063.295,388.462,-112.442,174.849,36.429,156.853
C00721=1063.302,388.708,-112.483,174.854,36.436,156.854
C00722=1063.310,388.955,-112.523,174.860,36.443,156.856
C00723=1063.317,389.202,-112.564,174.865,36.450,156.858
C00724=1063.325,389.448,-112.605,174.870,36.458,156.860
C00725=1063.332,389.694,-112.646,174.876,36.465,156.861
C00726=1063.340,389.941,-112.687,174.881,36.472,156.863
C00727=1063.347,390.187,-112.728,174.887,36.480,156.865
C00728=1063.355,390.434,-112.769,174.892,36.487,156.867
C00729=1063.363,390.680,-112.810,174.898,36.495,156.868
C00730=1063.370,390.927,-112.851,174.904,36.502,156.870
C00731=1063.378,391.173,-112.892,174.909,36.509,156.872
C00732=1063.385,391.420,-112.933,174.915,36.517,156.874
C00733=1063.393,391.666,-112.974,174.920,36.525,156.876
C00734=1063.401,391.913,-113.015,174.926,36.532,156.877
C00735=1063.408,392.159,-113.056,174.931,36.539,156.879
C00736=1063.416,392.405,-113.098,174.937,36.547,156.881
C00737=1063.423,392.652,-113.139,174.942,36.555,156.883
C00738=1063.431,392.898,-113.180,174.948,36.562,156.885
C00739=1063.438,393.145,-113.221,174.953,36.570,156.887
C00740=1063.446,393.391,-113.263,174.960,36.577,156.889
C00741=1063.453,393.637,-113.304,174.965,36.585,156.890
C00742=1063.461,393.883,-113.346,174.970,36.593,156.892
C00743=1063.469,394.129,-113.387,174.976,36.600,156.894
C00744=1063.476,394.376,-113.428,174.981,36.608,156.896
C00745=1063.484,394.622,-113.470,174.987,36.615,156.898
C00746=1063.491,394.869,-113.511,174.993,36.623,156.900
C00747=1063.498,395.115,-113.553,174.999,36.631,156.902
C00748=1063.506,395.362,-113.595,175.005,36.639,156.904
C00749=1063.514,395.608,-113.637,175.010,36.646,156.905
C00750=1063.521,395.854,-113.679,175.016,36.654,156.907
C00751=1063.529,396.100,-113.720,175.021,36.662,156.909
C00752=1063.536,396.346,-113.762,175.027,36.670,156.911
C00753=1063.544,396.592,-113.804,175.033,36.678,156.913
C00754=1063.552,396.840,-113.845,175.039,36.686,156.915
C00755=1063.559,397.086,-113.887,175.045,36.693,156.917
C00756=1063.568,397.331,-113.929,175.050,36.702,156.919
C00757=1063.576,397.578,-113.971,175.056,36.709,156.921
C00758=1063.583,397.825,-114.013,175.062,36.717,156.923
C00759=1063.590,398.071,-114.055,175.068,36.725,156.925
C00760=1063.598,398.317,-114.097,175.074,36.733,156.927
C00761=1063.606,398.563,-114.139,175.079,36.742,156.929
C00762=1063.613,398.809,-114.181,175.086,36.750,156.931
C00763=1063.622,399.056,-114.223,175.091,36.757,156.933
C00764=1063.629,399.302,-114.265,175.097,36.765,156.935
C00765=1063.636,399.548,-114.308,175.103,36.774,156.937
C00766=1063.644,399.795,-114.350,175.109,36.782,156.939
C00767=1063.652,400.041,-114.392,175.115,36.790,156.941
C00768=1063.660,400.288,-114.434,175.121,36.798,156.943
C00769=1063.670,400.609,-114.490,175.129,36.809,156.946
C00770=1063.681,400.931,-114.545,175.137,36.820,156.948
C00771=1063.691,401.253,-114.601,175.144,36.831,156.951
C00772=1063.701,401.575,-114.656,175.152,36.841,156.954
C00773=1063.709,401.822,-114.699,175.158,36.849,156.956
C00774=1063.716,402.068,-114.741,175.165,36.858,156.958
C00775=1063.724,402.314,-114.783,175.171,36.866,156.960
C00776=1063.733,402.560,-114.826,175.176,36.875,156.962
C00777=1063.740,402.807,-114.869,175.183,36.883,156.964
C00778=1063.748,403.053,-114.912,175.189,36.891,156.966
C00779=1063.756,403.299,-114.954,175.196,36.900,156.968
C00780=1063.764,403.545,-114.998,175.201,36.908,156.970
C00781=1063.772,403.792,-115.040,175.207,36.917,156.972
C00782=1063.779,404.037,-115.083,175.214,36.925,156.975
C00783=1063.787,404.284,-115.125,175.220,36.934,156.977
C00784=1063.796,404.530,-115.169,175.227,36.942,156.979
C00785=1063.803,404.776,-115.212,175.233,36.951,156.981
C00786=1063.811,405.022,-115.255,175.238,36.959,156.983
C00787=1063.819,405.269,-115.298,175.245,36.968,156.985
C00788=1063.827,405.514,-115.340,175.251,36.977,156.987
C00789=1063.835,405.760,-115.384,175.258,36.985,156.990
C00790=1063.843,406.006,-115.427,175.264,36.994,156.992
C00791=1063.851,406.253,-115.471,175.271,37.003,156.994
C00792=1063.858,406.499,-115.514,175.277,37.011,156.996
C00793=1063.866,406.745,-115.556,175.283,37.020,156.999
C00794=1063.874,406.992,-115.600,175.289,37.029,157.001
C00795=1063.883,407.237,-115.644,175.296,37.038,157.003
C00796=1063.891,407.483,-115.687,175.302,37.047,157.005
C00797=1063.898,407.729,-115.730,175.309,37.056,157.007
C00798=1063.906,407.975,-115.773,175.315,37.065,157.010
C00799=1063.914,408.221,-115.817,175.322,37.073,157.012
C00800=1063.922,408.468,-115.861,175.328,37.082,157.014
C00801=1063.930,408.714,-115.904,175.335,37.091,157.017
C00802=1063.938,408.960,-115.948,175.341,37.101,157.019
C00803=1063.946,409.206,-115.992,175.348,37.110,157.021
C00804=1063.955,409.452,-116.035,175.354,37.119,157.023
C00805=1063.963,409.698,-116.079,175.361,37.128,157.026
C00806=1063.970,409.944,-116.123,175.367,37.137,157.028
C00807=1063.978,410.190,-116.166,175.374,37.146,157.030
C00808=1063.987,410.436,-116.210,175.381,37.155,157.033
C00809=1063.995,410.682,-116.254,175.387,37.164,157.035
C00810=1064.003,410.928,-116.298,175.394,37.173,157.037
C00811=1064.011,411.174,-116.341,175.400,37.183,157.040
C00812=1064.019,411.420,-116.385,175.408,37.192,157.042
C00813=1064.027,411.666,-116.429,175.415,37.201,157.044
C00814=1064.035,411.912,-116.473,175.421,37.210,157.047
C00815=1064.044,412.157,-116.517,175.428,37.219,157.049
C00816=1064.052,412.404,-116.561,175.435,37.229,157.052
C00817=1064.060,412.650,-116.605,175.441,37.238,157.054
C00818=1064.068,412.896,-116.650,175.448,37.247,157.056
C00819=1064.077,413.142,-116.694,175.456,37.257,157.059
C00820=1064.085,413.387,-116.738,175.462,37.266,157.061
C00821=1064.093,413.613,-116.779,175.469,37.275,157.063
C00822=1064.101,413.838,-116.819,175.474,37.283,157.066
C00823=1064.108,414.063,-116.859,175.481,37.292,157.068
C00824=1064.116,414.288,-116.900,175.488,37.301,157.070
C00825=1064.126,414.594,-116.955,175.496,37.312,157.073
C00826=1064.136,414.900,-117.010,175.505,37.325,157.076
C00827=1064.147,415.206,-117.066,175.513,37.337,157.079
C00828=1064.157,415.512,-117.121,175.522,37.348,157.082
C00829=1064.165,415.758,-117.166,175.529,37.358,157.085
C00830=1064.173,416.003,-117.211,175.537,37.368,157.087
C00831=1064.181,416.250,-117.256,175.544,37.378,157.090
C00832=1064.190,416.495,-117.300,175.551,37.387,157.093
C00833=1064.199,416.741,-117.346,175.558,37.397,157.095
C00834=1064.207,416.987,-117.390,175.565,37.407,157.098
C00835=1064.215,417.233,-117.434,175.572,37.417,157.100
C00836=1064.224,417.479,-117.480,175.580,37.427,157.103
C00837=1064.232,417.724,-117.524,175.587,37.437,157.105
C00838=1064.241,417.970,-117.570,175.594,37.447,157.108
C00839=1064.249,418.216,-117.614,175.602,37.457,157.111
C00840=1064.257,418.462,-117.660,175.609,37.467,157.113
C00841=1064.265,418.707,-117.705,175.616,37.477,157.116
C00842=1064.274,418.954,-117.750,175.623,37.487,157.119
C00843=1064.282,419.199,-117.795,175.631,37.497,157.121
C00844=1064.291,419.444,-117.840,175.638,37.507,157.124
C00845=1064.300,419.691,-117.885,175.646,37.517,157.127
C00846=1064.308,419.936,-117.930,175.653,37.527,157.129
C00847=1064.317,420.182,-117.976,175.661,37.538,157.132
C00848=1064.326,420.428,-118.021,175.668,37.548,157.135
C00849=1064.334,420.673,-118.066,175.676,37.558,157.137
C00850=1064.342,420.919,-118.112,175.683,37.568,157.140
C00851=1064.351,421.165,-118.158,175.691,37.579,157.143
C00852=1064.360,421.410,-118.203,175.698,37.589,157.145
C00853=1064.368,421.656,-118.249,175.706,37.600,157.148
C00854=1064.377,421.902,-118.294,175.713,37.610,157.151
C00855=1064.385,422.147,-118.341,175.721,37.621,157.154
C00856=1064.394,422.393,-118.386,175.729,37.631,157.156
C00857=1064.402,422.639,-118.432,175.737,37.642,157.159
C00858=1064.411,422.885,-118.477,175.745,37.652,157.162
C00859=1064.420,423.129,-118.523,175.753,37.663,157.165
C00860=1064.428,423.375,-118.569,175.760,37.674,157.168
C00861=1064.437,423.621,-118.615,175.768,37.684,157.170
C00862=1064.445,423.867,-118.661,175.776,37.695,157.173
C00863=1064.454,424.113,-118.707,175.783,37.705,157.176
C00864=1064.463,424.358,-118.754,175.792,37.716,157.179
C00865=1064.472,424.604,-118.799,175.800,37.727,157.182
C00866=1064.480,424.849,-118.846,175.808,37.738,157.185
C00867=1064.490,425.095,-118.892,175.815,37.749,157.188
C00868=1064.497,425.340,-118.937,175.823,37.760,157.191
C00869=1064.507,425.585,-118.984,175.832,37.770,157.194
C00870=1064.515,425.831,-119.030,175.840,37.781,157.196
C00871=1064.525,426.077,-119.077,175.848,37.792,157.199
C00872=1064.534,426.322,-119.124,175.855,37.803,157.202
C00873=1064.543,426.568,-119.169,175.864,37.814,157.205
C00874=1064.551,426.814,-119.216,175.872,37.825,157.208
C00875=1064.560,427.059,-119.262,175.880,37.836,157.211
C00876=1064.569,427.304,-119.309,175.888,37.847,157.214
C00877=1064.578,427.550,-119.355,175.897,37.859,157.217
C00878=1064.586,427.795,-119.402,175.905,37.870,157.220
C00879=1064.596,428.040,-119.449,175.914,37.881,157.223
C00880=1064.604,428.285,-119.496,175.922,37.892,157.226
C00881=1064.616,428.612,-119.557,175.933,37.907,157.230
C00882=1064.627,428.938,-119.620,175.943,37.923,157.235
C00883=1064.640,429.264,-119.683,175.955,37.938,157.239
C00884=1064.652,429.589,-119.745,175.966,37.953,157.243
C00885=1064.661,429.835,-119.792,175.974,37.964,157.246
C00886=1064.670,430.080,-119.840,175.984,37.976,157.249
C00887=1064.679,430.326,-119.886,175.992,37.988,157.252
C00888=1064.688,430.571,-119.934,176.001,37.999,157.255
C00889=1064.697,430.817,-119.980,176.009,38.011,157.259
C00890=1064.706,431.062,-120.028,176.018,38.022,157.262
C00891=1064.715,431.307,-120.076,176.026,38.034,157.265
C00892=1064.724,431.553,-120.122,176.035,38.046,157.268
C00893=1064.733,431.798,-120.170,176.044,38.058,157.271
C00894=1064.742,432.043,-120.218,176.052,38.070,157.275
C00895=1064.751,432.288,-120.265,176.062,38.081,157.278
C00896=1064.760,432.534,-120.313,176.070,38.093,157.281
C00897=1064.769,432.779,-120.360,176.079,38.105,157.284
C00898=1064.779,433.024,-120.408,176.088,38.118,157.288
C00899=1064.788,433.269,-120.456,176.097,38.129,157.291
C00900=1064.797,433.515,-120.503,176.106,38.141,157.294
C00901=1064.806,433.759,-120.552,176.115,38.153,157.298
C00902=1064.816,434.004,-120.599,176.124,38.166,157.301
C00903=1064.825,434.249,-120.647,176.133,38.178,157.304
C00904=1064.834,434.495,-120.695,176.142,38.190,157.308
C00905=1064.843,434.740,-120.744,176.151,38.202,157.311
C00906=1064.852,434.985,-120.791,176.161,38.215,157.314
C00907=1064.861,435.231,-120.839,176.169,38.227,157.318
C00908=1064.871,435.476,-120.888,176.179,38.239,157.321
C00909=1064.880,435.720,-120.936,176.188,38.251,157.325
C00910=1064.890,435.966,-120.983,176.197,38.264,157.328
C00911=1064.899,436.211,-121.032,176.207,38.276,157.332
C00912=1064.909,436.456,-121.080,176.216,38.289,157.335
C00913=1064.918,436.700,-121.128,176.226,38.301,157.339
C00914=1064.927,436.946,-121.177,176.234,38.314,157.342
C00915=1064.937,437.191,-121.226,176.244,38.326,157.346
C00916=1064.946,437.436,-121.273,176.253,38.339,157.349
C00917=1064.956,437.681,-121.322,176.263,38.352,157.353
C00918=1064.966,437.926,-121.371,176.273,38.365,157.356
C00919=1064.976,438.171,-121.419,176.282,38.377,157.360
C00920=1064.985,438.416,-121.468,176.292,38.390,157.363
C00921=1064.994,438.661,-121.517,176.301,38.403,157.367
C00922=1065.004,438.906,-121.567,176.312,38.416,157.371
C00923=1065.013,439.151,-121.615,176.322,38.429,157.374
C00924=1065.023,439.396,-121.664,176.331,38.442,157.378
C00925=1065.032,439.641,-121.713,176.341,38.455,157.382
C00926=1065.042,439.886,-121.762,176.351,38.468,157.385
C00927=1065.052,440.131,-121.810,176.360,38.481,157.389
C00928=1065.061,440.376,-121.860,176.370,38.494,157.393
C00929=1065.071,440.620,-121.909,176.381,38.508,157.397
C00930=1065.080,440.865,-121.959,176.391,38.521,157.400
C00931=1065.090,441.110,-122.007,176.401,38.534,157.404
C00932=1065.100,441.355,-122.057,176.410,38.548,157.408
C00933=1065.110,441.600,-122.107,176.421,38.561,157.412
C00934=1065.119,441.845,-122.156,176.431,38.574,157.416
C00935=1065.129,442.089,-122.205,176.441,38.588,157.419
C00936=1065.139,442.335,-122.255,176.452,38.602,157.423
C00937=1065.156,442.743,-122.338,176.468,38.624,157.430
C00938=1065.172,443.152,-122.421,176.486,38.647,157.436
C00939=1065.189,443.560,-122.504,176.504,38.670,157.443
C00940=1065.205,443.969,-122.587,176.522,38.693,157.449
C00941=1065.215,444.214,-122.637,176.532,38.707,157.453
C00942=1065.225,444.458,-122.687,176.543,38.721,157.457
C00943=1065.235,444.703,-122.737,176.553,38.735,157.461
C00944=1065.244,444.948,-122.787,176.564,38.749,157.466
C00945=1065.255,445.192,-122.837,176.574,38.763,157.470
C00946=1065.265,445.437,-122.887,176.585,38.777,157.474
C00947=1065.275,445.682,-122.938,176.596,38.791,157.478
C00948=1065.284,445.926,-122.989,176.607,38.805,157.482
C00949=1065.295,446.171,-123.038,176.618,38.820,157.486
C00950=1065.305,446.415,-123.089,176.629,38.834,157.490
C00951=1065.315,446.660,-123.140,176.639,38.848,157.494
C00952=1065.326,446.904,-123.190,176.651,38.862,157.498
C00953=1065.336,447.148,-123.241,176.662,38.877,157.503
C00954=1065.346,447.392,-123.291,176.673,38.891,157.507
C00955=1065.356,447.637,-123.342,176.685,38.906,157.511
C00956=1065.367,447.881,-123.392,176.695,38.920,157.515
C00957=1065.378,448.124,-123.441,176.707,38.934,157.519
C00958=1065.391,448.368,-123.490,176.718,38.948,157.524
C00959=1065.404,448.612,-123.539,176.729,38.961,157.527
C00960=1065.420,448.858,-123.586,176.741,38.975,157.531
C00961=1065.435,449.103,-123.633,176.753,38.988,157.535
C00962=1065.452,449.347,-123.680,176.764,39.000,157.539
C00963=1065.470,449.593,-123.725,176.775,39.012,157.543
C00964=1065.488,449.838,-123.770,176.786,39.024,157.546
C00965=1065.149,449.843,-124.036,176.777,39.149,157.580
C00966=1065.130,449.598,-123.991,176.766,39.138,157.577
C00967=1065.112,449.353,-123.946,176.755,39.126,157.573
C00968=1065.095,449.107,-123.899,176.743,39.113,157.569
C00969=1065.079,448.863,-123.853,176.732,39.100,157.565
C00970=1065.064,448.617,-123.805,176.720,39.087,157.561
C00971=1065.050,448.373,-123.756,176.709,39.074,157.558
C00972=1065.037,448.130,-123.707,176.697,39.060,157.553
C00973=1065.026,447.886,-123.658,176.685,39.046,157.549
C00974=1065.015,447.642,-123.608,176.674,39.032,157.545
C00975=1065.004,447.397,-123.557,176.663,39.018,157.541
C00976=1064.995,447.153,-123.507,176.651,39.003,157.537
C00977=1064.984,446.910,-123.456,176.641,38.989,157.532
C00978=1064.974,446.666,-123.405,176.629,38.974,157.528
C00979=1064.964,446.420,-123.355,176.618,38.960,157.524
C00980=1064.954,446.176,-123.304,176.607,38.946,157.520
C00981=1064.943,445.932,-123.254,176.596,38.932,157.516
C00982=1064.933,445.687,-123.203,176.585,38.918,157.512
C00983=1064.924,445.442,-123.153,176.574,38.904,157.508
C00984=1064.913,445.198,-123.103,176.563,38.890,157.503
C00985=1064.903,444.953,-123.053,176.553,38.876,157.499
C00986=1064.893,444.709,-123.002,176.542,38.862,157.495
C00987=1064.883,444.463,-122.952,176.531,38.848,157.491
C00988=1064.873,444.219,-122.902,176.520,38.834,157.487
C00989=1064.863,443.975,-122.852,176.509,38.820,157.483
C00990=1064.848,443.585,-122.773,176.492,38.798,157.477
C00991=1064.831,443.196,-122.693,176.476,38.776,157.471
C00992=1064.815,442.806,-122.614,176.459,38.754,157.464
C00993=1064.800,442.417,-122.535,176.443,38.733,157.458
C00994=1064.790,442.172,-122.485,176.432,38.719,157.454
C00995=1064.780,441.927,-122.436,176.422,38.706,157.450
C00996=1064.770,441.682,-122.387,176.411,38.692,157.447
C00997=1064.761,441.438,-122.337,176.401,38.679,157.443
C00998=1064.750,441.193,-122.287,176.391,38.666,157.439
C00999=1064.741,440.947,-122.238,176.380,38.652,157.435
C01000=1064.731,440.703,-122.189,176.371,38.639,157.431
C01001=1064.722,440.458,-122.139,176.361,38.626,157.428
C01002=1064.712,440.213,-122.091,176.351,38.613,157.424
C01003=1064.702,439.968,-122.040,176.340,38.600,157.420
C01004=1064.693,439.723,-121.992,176.331,38.587,157.416
C01005=1064.683,439.478,-121.943,176.321,38.574,157.413
C01006=1064.673,439.233,-121.894,176.311,38.561,157.409
C01007=1064.664,438.988,-121.845,176.302,38.548,157.405
C01008=1064.655,438.743,-121.796,176.291,38.535,157.402
C01009=1064.645,438.499,-121.747,176.281,38.522,157.398
C01010=1064.635,438.254,-121.698,176.272,38.509,157.395
C01011=1064.626,438.008,-121.649,176.262,38.497,157.391
C01012=1064.616,437.763,-121.601,176.252,38.484,157.387
C01013=1064.606,437.519,-121.552,176.243,38.471,157.384
C01014=1064.597,437.274,-121.503,176.233,38.458,157.380
C01015=1064.587,437.028,-121.456,176.224,38.446,157.377
C01016=1064.577,436.783,-121.407,176.214,38.434,157.373
C01017=1064.568,436.539,-121.359,176.205,38.421,157.370
C01018=1064.559,436.293,-121.310,176.195,38.409,157.366
C01019=1064.550,436.048,-121.262,176.186,38.396,157.363
C01020=1064.540,435.803,-121.213,176.176,38.383,157.359
C01021=1064.530,435.558,-121.165,176.167,38.371,157.356
C01022=1064.521,435.313,-121.118,176.157,38.359,157.352
C01023=1064.512,435.068,-121.069,176.149,38.347,157.349
C01024=1064.502,434.822,-121.021,176.140,38.334,157.346
C01025=1064.493,434.578,-120.973,176.130,38.322,157.342
C01026=1064.484,434.333,-120.925,176.121,38.310,157.339
C01027=1064.474,434.087,-120.877,176.111,38.298,157.335
C01028=1064.466,433.842,-120.829,176.102,38.286,157.332
C01029=1064.456,433.597,-120.781,176.094,38.273,157.329
C01030=1064.447,433.351,-120.733,176.085,38.262,157.325
C01031=1064.438,433.106,-120.686,176.075,38.250,157.322
C01032=1064.428,432.861,-120.638,176.066,38.237,157.319
C01033=1064.419,432.616,-120.590,176.058,38.226,157.315
C01034=1064.410,432.371,-120.542,176.049,38.214,157.312
C01035=1064.401,432.126,-120.494,176.039,38.202,157.309
C01036=1064.392,431.881,-120.447,176.031,38.190,157.306
C01037=1064.383,431.635,-120.400,176.022,38.178,157.302
C01038=1064.374,431.390,-120.352,176.013,38.166,157.299
C01039=1064.365,431.144,-120.305,176.005,38.155,157.296
C01040=1064.356,430.899,-120.257,175.996,38.143,157.293
C01041=1064.346,430.654,-120.209,175.986,38.131,157.289
C01042=1064.338,430.408,-120.163,175.978,38.120,157.286
C01043=1064.328,430.164,-120.116,175.969,38.108,157.283
C01044=1064.319,429.918,-120.069,175.961,38.097,157.280
C01045=1064.310,429.673,-120.021,175.952,38.086,157.277
C01046=1064.298,429.345,-119.958,175.941,38.070,157.273
C01047=1064.286,429.017,-119.895,175.930,38.055,157.269
C01048=1064.274,428.689,-119.832,175.918,38.040,157.264
C01049=1064.263,428.361,-119.771,175.907,38.025,157.260
C01050=1064.253,428.117,-119.724,175.899,38.014,157.257
C01051=1064.244,427.871,-119.677,175.890,38.002,157.254
C01052=1064.236,427.626,-119.630,175.882,37.991,157.251
C01053=1064.227,427.379,-119.583,175.873,37.980,157.248
C01054=1064.217,427.134,-119.537,175.865,37.969,157.245
C01055=1064.209,426.889,-119.490,175.858,37.958,157.242
C01056=1064.200,426.643,-119.444,175.849,37.947,157.239
C01057=1064.191,426.398,-119.397,175.841,37.935,157.236
C01058=1064.183,426.152,-119.351,175.832,37.924,157.233
C01059=1064.173,425.907,-119.305,175.824,37.914,157.230
C01060=1064.165,425.662,-119.258,175.816,37.903,157.227
C01061=1064.155,425.416,-119.212,175.808,37.892,157.224
C01062=1064.147,425.170,-119.166,175.800,37.881,157.221
C01063=1064.138,424.925,-119.120,175.792,37.870,157.219
C01064=1064.129,424.680,-119.073,175.784,37.859,157.216
C01065=1064.120,424.434,-119.027,175.776,37.849,157.213
C01066=1064.112,424.188,-118.981,175.768,37.838,157.210
C01067=1064.103,423.943,-118.934,175.760,37.827,157.207
C01068=1064.094,423.697,-118.888,175.752,37.817,157.204
C01069=1064.085,423.452,-118.842,175.744,37.806,157.201
C01070=1064.076,423.206,-118.797,175.737,37.795,157.199
C01071=1064.068,422.960,-118.751,175.728,37.785,157.196
C01072=1064.059,422.715,-118.705,175.720,37.775,157.193
C01073=1064.051,422.469,-118.659,175.713,37.764,157.190
C01074=1064.042,422.223,-118.614,175.705,37.753,157.187
C01075=1064.033,421.978,-118.567,175.698,37.743,157.185
C01076=1064.025,421.733,-118.522,175.690,37.732,157.182
C01077=1064.017,421.487,-118.476,175.682,37.722,157.179
C01078=1064.008,421.241,-118.431,175.675,37.712,157.176
C01079=1063.999,420.995,-118.385,175.666,37.701,157.174
C01080=1063.991,420.749,-118.339,175.659,37.691,157.171
C01081=1063.982,420.504,-118.294,175.651,37.681,157.168
C01082=1063.973,420.258,-118.249,175.644,37.670,157.165
C01083=1063.965,420.013,-118.204,175.636,37.660,157.163
C01084=1063.957,419.767,-118.158,175.629,37.650,157.160
C01085=1063.948,419.521,-118.112,175.621,37.640,157.157
C01086=1063.939,419.276,-118.067,175.614,37.630,157.155
C01087=1063.931,419.029,-118.022,175.606,37.620,157.152
C01088=1063.922,418.784,-117.977,175.599,37.610,157.149
C01089=1063.913,418.538,-117.932,175.591,37.600,157.147
C01090=1063.904,418.292,-117.886,175.584,37.590,157.144
C01091=1063.897,418.046,-117.842,175.576,37.580,157.142
C01092=1063.888,417.800,-117.796,175.570,37.570,157.139
C01093=1063.880,417.555,-117.752,175.562,37.560,157.136
C01094=1063.871,417.309,-117.706,175.555,37.550,157.134
C01095=1063.863,417.063,-117.662,175.548,37.540,157.131
C01096=1063.854,416.818,-117.617,175.540,37.531,157.129
C01097=1063.846,416.572,-117.572,175.533,37.521,157.126
C01098=1063.837,416.326,-117.527,175.526,37.511,157.124
C01099=1063.829,416.080,-117.483,175.518,37.501,157.121
C01100=1063.821,415.834,-117.438,175.511,37.492,157.118
C01101=1063.813,415.588,-117.393,175.505,37.482,157.116
C01102=1063.802,415.281,-117.337,175.495,37.469,157.113
C01103=1063.792,414.973,-117.281,175.487,37.457,157.110
C01104=1063.782,414.664,-117.226,175.478,37.446,157.106
C01105=1063.772,414.357,-117.170,175.468,37.434,157.103
C01106=1063.763,414.111,-117.125,175.462,37.424,157.101
C01107=1063.754,413.865,-117.081,175.455,37.414,157.098
C01108=1063.746,413.619,-117.037,175.448,37.405,157.096
C01109=1063.738,413.373,-116.992,175.441,37.396,157.094
C01110=1063.730,413.127,-116.948,175.434,37.386,157.091
C01111=1063.722,412.881,-116.904,175.427,37.377,157.089
C01112=1063.712,412.635,-116.860,175.420,37.368,157.086
C01113=1063.704,412.389,-116.816,175.413,37.358,157.084
C01114=1063.696,412.143,-116.772,175.407,37.349,157.082
C01115=1063.688,411.898,-116.727,175.399,37.340,157.079
C01116=1063.680,411.651,-116.684,175.392,37.331,157.077
C01117=1063.672,411.406,-116.640,175.386,37.321,157.074
C01118=1063.663,411.159,-116.595,175.379,37.312,157.072
C01119=1063.655,410.913,-116.552,175.372,37.303,157.070
C01120=1063.646,410.667,-116.508,175.366,37.294,157.067
C01121=1063.639,410.421,-116.464,175.359,37.285,157.065
C01122=1063.631,410.175,-116.420,175.352,37.276,157.063
C01123=1063.622,409.929,-116.377,175.346,37.267,157.060
C01124=1063.614,409.684,-116.333,175.339,37.257,157.058
C01125=1063.606,409.437,-116.289,175.333,37.248,157.056
C01126=1063.598,409.191,-116.246,175.326,37.239,157.053
C01127=1063.590,408.945,-116.202,175.319,37.230,157.051
C01128=1063.582,408.699,-116.158,175.313,37.222,157.049
C01129=1063.574,408.453,-116.114,175.306,37.213,157.047
C01130=1063.565,408.207,-116.071,175.300,37.204,157.044
C01131=1063.558,407.962,-116.027,175.293,37.195,157.042
C01132=1063.550,407.715,-115.984,175.287,37.186,157.040
C01133=1063.542,407.469,-115.941,175.280,37.177,157.037
C01134=1063.534,407.223,-115.897,175.273,37.168,157.035
C01135=1063.526,406.977,-115.854,175.267,37.159,157.033
C01136=1063.518,406.730,-115.810,175.260,37.151,157.031
C01137=1063.511,406.485,-115.767,175.254,37.142,157.028
C01138=1063.502,406.239,-115.724,175.247,37.133,157.026
C01139=1063.494,405.992,-115.681,175.241,37.124,157.024
C01140=1063.487,405.746,-115.637,175.235,37.116,157.022
C01141=1063.478,405.500,-115.594,175.229,37.107,157.020
C01142=1063.470,405.255,-115.551,175.222,37.098,157.018
C01143=1063.463,405.008,-115.508,175.216,37.090,157.015
C01144=1063.454,404.761,-115.465,175.209,37.081,157.013
C01145=1063.447,404.515,-115.422,175.203,37.073,157.011
C01146=1063.439,404.270,-115.379,175.196,37.064,157.009
C01147=1063.431,404.023,-115.336,175.191,37.056,157.007
C01148=1063.423,403.777,-115.293,175.185,37.047,157.005
C01149=1063.415,403.531,-115.250,175.178,37.038,157.002
C01150=1063.407,403.284,-115.207,175.172,37.030,157.000
C01151=1063.399,403.039,-115.165,175.166,37.022,156.998
C01152=1063.392,402.792,-115.122,175.160,37.013,156.996
C01153=1063.384,402.546,-115.079,175.154,37.005,156.994
C01154=1063.374,402.250,-115.028,175.146,36.995,156.991
C01155=1063.364,401.953,-114.977,175.139,36.985,156.989
C01156=1063.355,401.656,-114.926,175.132,36.975,156.986
C01157=1063.345,401.360,-114.874,175.124,36.965,156.984
C01158=1063.337,401.107,-114.830,175.118,36.957,156.982
C01159=1063.330,400.855,-114.787,175.111,36.948,156.980
C01160=1063.321,400.602,-114.744,175.106,36.940,156.978
C01161=1063.314,400.349,-114.700,175.099,36.932,156.976
C01162=1063.306,400.104,-114.658,175.093,36.923,156.974
C01163=1063.298,399.857,-114.615,175.087,36.915,156.972
C01164=1063.290,399.611,-114.573,175.081,36.907,156.970
C01165=1063.282,399.365,-114.531,175.075,36.899,156.968
C01166=1063.275,399.119,-114.489,175.069,36.891,156.966
C01167=1063.267,398.873,-114.447,175.064,36.883,156.964
C01168=1063.259,398.626,-114.404,175.057,36.875,156.962
C01169=1063.251,398.380,-114.362,175.052,36.867,156.960
C01170=1063.244,398.134,-114.320,175.046,36.859,156.957
C01171=1063.236,397.887,-114.278,175.039,36.851,156.956
C01172=1063.229,397.641,-114.236,175.034,36.843,156.954
C01173=1063.221,397.395,-114.194,175.028,36.835,156.952
C01174=1063.213,397.148,-114.152,175.023,36.827,156.950
C01175=1063.205,396.902,-114.111,175.016,36.819,156.948
C01176=1063.197,396.656,-114.069,175.010,36.811,156.946
C01177=1063.189,396.409,-114.027,175.005,36.804,156.944
C01178=1063.182,396.163,-113.985,174.999,36.796,156.942
C01179=1063.174,395.917,-113.943,174.993,36.788,156.940
C01180=1063.167,395.671,-113.901,174.987,36.780,156.938
C01181=1063.159,395.424,-113.860,174.982,36.772,156.936
C01182=1063.151,395.178,-113.818,174.976,36.765,156.934
C01183=1063.144,394.931,-113.777,174.970,36.757,156.932
C01184=1063.136,394.685,-113.735,174.964,36.750,156.931
C01185=1063.129,394.439,-113.693,174.958,36.741,156.929
C01186=1063.122,394.192,-113.651,174.953,36.734,156.927
C01187=1063.114,393.946,-113.610,174.947,36.726,156.925
C01188=1063.106,393.700,-113.569,174.942,36.719,156.923
C01189=1063.099,393.454,-113.528,174.936,36.711,156.921
C01190=1063.090,393.207,-113.485,174.930,36.703,156.919
C01191=1063.083,392.960,-113.444,174.924,36.696,156.917
C01192=1063.076,392.714,-113.403,174.919,36.688,156.915
C01193=1063.068,392.468,-113.362,174.913,36.681,156.914
C01194=1063.060,392.221,-113.320,174.908,36.674,156.912
C01195=1063.053,391.975,-113.279,174.903,36.666,156.910
C01196=1063.045,391.729,-113.238,174.897,36.658,156.908
C01197=1063.037,391.483,-113.197,174.891,36.651,156.906
C01198=1063.030,391.236,-113.155,174.885,36.644,156.905
C01199=1063.023,390.989,-113.114,174.880,36.636,156.903
C01200=1063.015,390.743,-113.073,174.874,36.628,156.901
C01201=1063.008,390.497,-113.033,174.869,36.621,156.899
C01202=1063.001,390.251,-112.991,174.864,36.614,156.897
C01203=1062.993,390.004,-112.951,174.858,36.607,156.896
C01204=1062.985,389.758,-112.909,174.853,36.599,156.894
C01205=1062.977,389.512,-112.869,174.847,36.592,156.892
C01206=1062.970,389.265,-112.828,174.842,36.585,156.890
C01207=1062.962,389.018,-112.788,174.837,36.578,156.889
C01208=1062.955,388.771,-112.746,174.830,36.570,156.887
C01209=1062.947,388.525,-112.706,174.825,36.563,156.885
C01210=1062.939,388.279,-112.665,174.819,36.556,156.883
C01211=1062.932,388.032,-112.624,174.814,36.549,156.882
C01212=1062.924,387.785,-112.584,174.809,36.542,156.880
C01213=1062.917,387.539,-112.543,174.803,36.535,156.878
C01214=1062.908,387.253,-112.496,174.797,36.526,156.876
C01215=1062.900,386.967,-112.448,174.791,36.518,156.874
C01216=1062.891,386.680,-112.402,174.785,36.509,156.872
C01217=1062.883,386.394,-112.355,174.778,36.501,156.870
C01218=1062.875,386.148,-112.314,174.773,36.494,156.868
C01219=1062.868,385.901,-112.274,174.768,36.487,156.867
C01220=1062.860,385.655,-112.233,174.762,36.480,156.865
C01221=1062.852,385.408,-112.193,174.757,36.473,156.863
C01222=1062.845,385.162,-112.152,174.752,36.466,156.862
C01223=1062.838,384.916,-112.113,174.747,36.459,156.860
C01224=1062.831,384.668,-112.072,174.742,36.452,156.858
C01225=1062.823,384.422,-112.031,174.737,36.445,156.857
C01226=1062.816,384.176,-111.992,174.732,36.438,156.855
C01227=1062.809,383.929,-111.951,174.727,36.432,156.853
C01228=1062.801,383.682,-111.911,174.721,36.424,156.852
C01229=1062.794,383.436,-111.871,174.716,36.417,156.850
C01230=1062.787,383.189,-111.831,174.711,36.411,156.848
C01231=1062.779,382.943,-111.790,174.706,36.404,156.847
C01232=1062.772,382.696,-111.750,174.700,36.397,156.845
C01233=1062.765,382.449,-111.710,174.695,36.390,156.843
C01234=1062.758,382.203,-111.670,174.690,36.383,156.842
C01235=1062.751,381.956,-111.630,174.685,36.376,156.840
C01236=1062.743,381.710,-111.590,174.680,36.369,156.839
C01237=1062.736,381.463,-111.550,174.675,36.363,156.837
C01238=1062.729,381.216,-111.510,174.669,36.356,156.835
C01239=1062.721,380.970,-111.470,174.664,36.349,156.834
C01240=1062.715,380.723,-111.431,174.659,36.343,156.832
C01241=1062.707,380.476,-111.391,174.654,36.336,156.831
C01242=1062.700,380.230,-111.351,174.650,36.329,156.829
C01243=1062.692,379.983,-111.311,174.645,36.322,156.827
C01244=1062.685,379.737,-111.272,174.639,36.316,156.826
C01245=1062.677,379.490,-111.232,174.634,36.309,156.824
C01246=1062.670,379.244,-111.192,174.629,36.302,156.823
C01247=1062.663,378.996,-111.153,174.624,36.296,156.821
C01248=1062.656,378.750,-111.113,174.619,36.290,156.820
C01249=1062.648,378.503,-111.073,174.614,36.283,156.818
C01250=1062.641,378.257,-111.034,174.609,36.276,156.816
C01251=1062.634,378.009,-110.994,174.604,36.270,156.815
C01252=1062.627,377.763,-110.955,174.599,36.263,156.813
C01253=1062.620,377.517,-110.915,174.594,36.256,156.812
C01254=1062.612,377.269,-110.876,174.589,36.250,156.810
C01255=1062.605,377.023,-110.836,174.584,36.244,156.809
C01256=1062.598,376.776,-110.798,174.579,36.237,156.807
C01257=1062.591,376.529,-110.758,174.574,36.230,156.806
C01258=1062.584,376.282,-110.719,174.570,36.224,156.804
C01259=1062.577,376.036,-110.679,174.565,36.218,156.803
C01260=1062.569,375.789,-110.640,174.560,36.211,156.801
C01261=1062.562,375.542,-110.601,174.555,36.205,156.800
C01262=1062.555,375.296,-110.562,174.550,36.198,156.798
C01263=1062.547,375.049,-110.522,174.545,36.192,156.797
C01264=1062.540,374.802,-110.484,174.541,36.186,156.795
C01265=1062.533,374.555,-110.445,174.536,36.180,156.794
C01266=1062.526,374.309,-110.405,174.531,36.173,156.792
C01267=1062.519,374.062,-110.366,174.526,36.167,156.791
C01268=1062.512,373.815,-110.327,174.521,36.160,156.789
C01269=1062.505,373.568,-110.288,174.517,36.154,156.788
C01270=1062.498,373.313,-110.248,174.511,36.147,156.786
C01271=1062.491,373.057,-110.207,174.506,36.141,156.785
C01272=1062.483,372.802,-110.167,174.501,36.135,156.783
C01273=1062.476,372.547,-110.126,174.496,36.128,156.782
C01274=1062.469,372.300,-110.088,174.491,36.122,156.780
C01275=1062.462,372.053,-110.049,174.487,36.115,156.779
C01276=1062.454,371.806,-110.010,174.482,36.109,156.777
C01277=1062.447,371.559,-109.971,174.477,36.103,156.776
C01278=1062.440,371.312,-109.932,174.472,36.097,156.774
C01279=1062.433,371.066,-109.894,174.468,36.091,156.773
C01280=1062.426,370.819,-109.855,174.463,36.085,156.771
C01281=1062.419,370.572,-109.817,174.458,36.078,156.770
C01282=1062.412,370.325,-109.779,174.453,36.072,156.769
C01283=1062.404,370.077,-109.740,174.449,36.066,156.767
C01284=1062.398,369.830,-109.701,174.445,36.060,156.766
C01285=1062.390,369.584,-109.663,174.440,36.054,156.764
C01286=1062.383,369.337,-109.624,174.435,36.048,156.763
C01287=1062.376,369.091,-109.586,174.431,36.042,156.762
C01288=1062.369,368.843,-109.548,174.426,36.036,156.760
C01289=1062.362,368.596,-109.509,174.421,36.030,156.759
C01290=1062.355,368.350,-109.470,174.416,36.024,156.757
C01291=1062.348,368.102,-109.432,174.412,36.018,156.756
C01292=1062.341,367.856,-109.394,174.407,36.012,156.755
C01293=1062.334,367.609,-109.355,174.402,36.006,156.753
C01294=1062.327,367.362,-109.317,174.398,36.000,156.752
C01295=1062.320,367.115,-109.279,174.394,35.994,156.750
C01296=1062.313,366.868,-109.240,174.389,35.988,156.749
C01297=1062.306,366.621,-109.203,174.384,35.982,156.748
C01298=1062.299,366.374,-109.164,174.380,35.976,156.746
C01299=1062.292,366.127,-109.126,174.375,35.970,156.745
C01300=1062.285,365.880,-109.087,174.370,35.964,156.744
C01301=1062.278,365.633,-109.049,174.367,35.958,156.742
C01302=1062.271,365.386,-109.011,174.362,35.952,156.741
C01303=1062.265,365.140,-108.973,174.357,35.947,156.740
C01304=1062.258,364.893,-108.936,174.352,35.941,156.738
C01305=1062.251,364.646,-108.897,174.348,35.935,156.737
C01306=1062.244,364.399,-108.859,174.343,35.929,156.736
C01307=1062.237,364.152,-108.820,174.339,35.923,156.734
C01308=1062.230,363.905,-108.783,174.335,35.917,156.733
C01309=1062.223,363.657,-108.745,174.330,35.911,156.732
C01310=1062.216,363.410,-108.707,174.325,35.906,156.730
C01311=1062.209,363.164,-108.670,174.321,35.900,156.729
C01312=1062.202,362.917,-108.631,174.317,35.894,156.728
C01313=1062.195,362.670,-108.594,174.312,35.888,156.726
C01314=1062.188,362.422,-108.556,174.308,35.883,156.725
C01315=1062.181,362.175,-108.518,174.303,35.877,156.724
C01316=1062.174,361.928,-108.481,174.298,35.871,156.722
C01317=1062.168,361.681,-108.443,174.295,35.865,156.721
C01318=1062.160,361.434,-108.406,174.290,35.860,156.720
C01319=1062.154,361.187,-108.368,174.285,35.854,156.718
C01320=1062.147,360.940,-108.330,174.281,35.849,156.717
C01321=1062.140,360.693,-108.293,174.277,35.843,156.716
C01322=1062.133,360.452,-108.256,174.273,35.837,156.715
C01323=1062.126,360.209,-108.219,174.268,35.832,156.713
C01324=1062.119,359.967,-108.182,174.264,35.826,156.712
C01325=1062.112,359.725,-108.146,174.260,35.820,156.711
C01326=1062.106,359.482,-108.109,174.255,35.815,156.710
C01327=1062.099,359.240,-108.072,174.251,35.810,156.708
C01328=1062.092,358.998,-108.036,174.247,35.804,156.707
C01329=1062.086,358.755,-107.999,174.242,35.798,156.706
C01330=1062.079,358.509,-107.962,174.239,35.793,156.705
C01331=1062.072,358.261,-107.924,174.234,35.788,156.703
C01332=1062.065,358.014,-107.887,174.229,35.782,156.702
C01333=1062.058,357.767,-107.850,174.226,35.777,156.701
C01334=1062.051,357.520,-107.813,174.221,35.771,156.700
C01335=1062.044,357.273,-107.775,174.217,35.765,156.698
C01336=1062.037,357.026,-107.739,174.212,35.760,156.697
C01337=1062.030,356.779,-107.701,174.208,35.755,156.696
C01338=1062.023,356.532,-107.664,174.204,35.749,156.695
C01339=1062.017,356.285,-107.627,174.199,35.744,156.693
C01340=1062.009,356.037,-107.590,174.196,35.738,156.692
C01341=1062.003,355.790,-107.553,174.191,35.732,156.691
C01342=1061.996,355.543,-107.516,174.186,35.727,156.690
C01343=1061.990,355.295,-107.478,174.183,35.722,156.688
C01344=1061.983,355.049,-107.441,174.178,35.716,156.687
C01345=1061.976,354.801,-107.404,174.175,35.711,156.686
C01346=1061.969,354.555,-107.367,174.170,35.705,156.685
C01347=1061.962,354.307,-107.331,174.166,35.700,156.684
C01348=1061.955,354.060,-107.294,174.162,35.695,156.682
C01349=1061.948,353.813,-107.257,174.157,35.690,156.681
C01350=1061.942,353.566,-107.220,174.153,35.684,156.680
C01351=1061.935,353.318,-107.184,174.149,35.679,156.679
C01352=1061.928,353.072,-107.146,174.145,35.673,156.678
C01353=1061.921,352.824,-107.110,174.141,35.668,156.676
C01354=1061.915,352.577,-107.073,174.137,35.662,156.675
C01355=1061.908,352.330,-107.036,174.132,35.657,156.674
C01356=1061.901,352.083,-106.999,174.128,35.652,156.673
C01357=1061.894,351.835,-106.962,174.124,35.646,156.672
C01358=1061.888,351.588,-106.926,174.120,35.641,156.670
C01359=1061.881,351.340,-106.889,174.116,35.636,156.669
C01360=1061.874,351.093,-106.853,174.111,35.631,156.668
C01361=1061.867,350.847,-106.816,174.108,35.625,156.667
C01362=1061.860,350.599,-106.779,174.103,35.620,156.666
C01363=1061.854,350.352,-106.743,174.100,35.615,156.664
C01364=1061.846,350.105,-106.707,174.095,35.610,156.663
C01365=1061.840,349.858,-106.670,174.092,35.604,156.662
C01366=1061.833,349.610,-106.633,174.087,35.599,156.661
C01367=1061.827,349.363,-106.597,174.082,35.594,156.660
C01368=1061.820,349.116,-106.561,174.079,35.589,156.659
C01369=1061.813,348.868,-106.524,174.074,35.584,156.658
C01370=1061.806,348.621,-106.488,174.071,35.578,156.656
C01371=1061.800,348.374,-106.452,174.066,35.573,156.655
C01372=1061.793,348.126,-106.416,174.063,35.568,156.654
C01373=1061.786,347.879,-106.379,174.058,35.563,156.653
C01374=1061.780,347.632,-106.343,174.055,35.558,156.652
C01375=1061.772,347.385,-106.307,174.050,35.553,156.651
C01376=1061.766,347.138,-106.270,174.047,35.548,156.650
C01377=1061.760,346.890,-106.235,174.042,35.542,156.648
C01378=1061.753,346.650,-106.199,174.039,35.537,156.647
C01379=1061.747,346.410,-106.165,174.034,35.533,156.646
C01380=1061.740,346.170,-106.129,174.031,35.528,156.645
C01381=1061.733,345.930,-106.094,174.027,35.523,156.644
C01382=1061.727,345.690,-106.059,174.023,35.518,156.643
C01383=1061.721,345.450,-106.024,174.019,35.513,156.642
C01384=1061.714,345.209,-105.989,174.015,35.508,156.641
C01385=1061.707,344.970,-105.954,174.011,35.503,156.640
C01386=1061.701,344.722,-105.919,174.008,35.498,156.639
C01387=1061.694,344.474,-105.882,174.003,35.493,156.637
C01388=1061.688,344.227,-105.847,174.000,35.488,156.636
C01389=1061.681,343.980,-105.810,173.995,35.483,156.635
C01390=1061.674,343.733,-105.775,173.992,35.477,156.634
C01391=1061.668,343.486,-105.739,173.987,35.473,156.633
C01392=1061.661,343.238,-105.703,173.984,35.468,156.632
C01393=1061.654,342.990,-105.667,173.979,35.463,156.631
C01394=1061.648,342.743,-105.631,173.976,35.457,156.630
C01395=1061.641,342.496,-105.596,173.972,35.453,156.629
C01396=1061.635,342.249,-105.560,173.968,35.448,156.628
C01397=1061.628,342.001,-105.525,173.965,35.443,156.627
C01398=1061.621,341.754,-105.488,173.960,35.438,156.625
C01399=1061.614,341.506,-105.453,173.957,35.433,156.624
C01400=1061.607,341.259,-105.418,173.952,35.428,156.623
C01401=1061.601,341.012,-105.381,173.949,35.423,156.622
C01402=1061.594,340.764,-105.346,173.945,35.419,156.621
C01403=1061.587,340.517,-105.311,173.941,35.413,156.620
C01404=1061.581,340.269,-105.275,173.937,35.408,156.619
C01405=1061.574,340.023,-105.239,173.933,35.404,156.618
C01406=1061.568,339.775,-105.204,173.929,35.398,156.617
C01407=1061.561,339.527,-105.168,173.926,35.394,156.616
C01408=1061.554,339.280,-105.133,173.921,35.389,156.615
C01409=1061.547,339.032,-105.098,173.918,35.384,156.614
C01410=1061.541,338.784,-105.062,173.915,35.379,156.613
C01411=1061.535,338.537,-105.027,173.910,35.374,156.612
C01412=1061.528,338.290,-104.991,173.907,35.369,156.610
C01413=1061.521,338.043,-104.955,173.902,35.365,156.609
C01414=1061.515,337.795,-104.920,173.899,35.359,156.608
C01415=1061.508,337.548,-104.885,173.895,35.355,156.607
C01416=1061.501,337.301,-104.850,173.891,35.350,156.606
C01417=1061.495,337.053,-104.814,173.887,35.345,156.605
C01418=1061.488,336.806,-104.779,173.884,35.341,156.604
C01419=1061.482,336.558,-104.744,173.880,35.336,156.603
C01420=1061.475,336.310,-104.710,173.876,35.331,156.602
C01421=1061.468,336.063,-104.675,173.873,35.326,156.601
C01422=1061.462,335.815,-104.639,173.868,35.322,156.600
C01423=1061.455,335.568,-104.604,173.865,35.316,156.599
C01424=1061.449,335.320,-104.569,173.861,35.312,156.598
C01425=1061.443,335.074,-104.534,173.857,35.307,156.597
C01426=1061.436,334.826,-104.499,173.854,35.303,156.596
C01427=1061.429,334.578,-104.464,173.850,35.298,156.595
C01428=1061.423,334.331,-104.429,173.846,35.293,156.594
C01429=1061.416,334.084,-104.394,173.842,35.288,156.593
C01430=1061.409,333.836,-104.359,173.839,35.284,156.592
C01431=1061.403,333.588,-104.324,173.836,35.279,156.591
C01432=1061.396,333.341,-104.289,173.831,35.274,156.590
C01433=1061.389,333.094,-104.254,173.828,35.269,156.589
C01434=1061.383,332.851,-104.220,173.824,35.265,156.588
C01435=1061.377,332.609,-104.187,173.821,35.260,156.587
C01436=1061.370,332.366,-104.153,173.817,35.256,156.586
C01437=1061.364,332.124,-104.118,173.813,35.251,156.585
C01438=1061.358,331.882,-104.084,173.810,35.247,156.584
C01439=1061.351,331.639,-104.050,173.806,35.242,156.583
C01440=1061.345,331.396,-104.016,173.803,35.237,156.582
C01441=1061.338,331.154,-103.982,173.799,35.233,156.581
C01442=1061.332,330.907,-103.947,173.795,35.228,156.580
C01443=1061.326,330.659,-103.913,173.792,35.224,156.579
C01444=1061.319,330.412,-103.878,173.788,35.219,156.578
C01445=1061.312,330.164,-103.844,173.784,35.214,156.577
C01446=1061.305,329.917,-103.809,173.781,35.210,156.576
C01447=1061.299,329.669,-103.774,173.777,35.205,156.575
C01448=1061.292,329.422,-103.741,173.774,35.200,156.574
C01449=1061.285,329.174,-103.706,173.769,35.196,156.573
C01450=1061.279,328.926,-103.671,173.766,35.192,156.572
C01451=1061.272,328.679,-103.637,173.763,35.187,156.571
C01452=1061.265,328.431,-103.602,173.759,35.182,156.570
C01453=1061.259,328.184,-103.568,173.755,35.178,156.569
C01454=1061.252,327.936,-103.534,173.752,35.174,156.568
C01455=1061.245,327.688,-103.500,173.748,35.169,156.567
C01456=1061.239,327.440,-103.465,173.745,35.165,156.566
C01457=1061.232,327.194,-103.431,173.740,35.160,156.565
C01458=1061.225,326.946,-103.397,173.737,35.156,156.564
C01459=1061.219,326.698,-103.362,173.734,35.151,156.563
C01460=1061.212,326.450,-103.329,173.730,35.147,156.562
C01461=1061.206,326.203,-103.295,173.727,35.142,156.561
C01462=1061.199,325.955,-103.261,173.723,35.138,156.561
C01463=1061.192,325.708,-103.226,173.719,35.133,156.560
C01464=1061.186,325.461,-103.192,173.716,35.129,156.559
C01465=1061.179,325.213,-103.158,173.712,35.124,156.558
C01466=1061.172,324.965,-103.123,173.709,35.120,156.557
C01467=1061.166,324.718,-103.090,173.706,35.115,156.556
C01468=1061.159,324.470,-103.055,173.701,35.111,156.555
C01469=1061.153,324.222,-103.021,173.698,35.106,156.554
C01470=1061.146,323.975,-102.988,173.695,35.102,156.553
C01471=1061.140,323.727,-102.953,173.691,35.097,156.552
C01472=1061.133,323.480,-102.920,173.688,35.093,156.551
C01473=1061.127,323.232,-102.885,173.685,35.088,156.550
C01474=1061.121,322.984,-102.852,173.681,35.084,156.549
C01475=1061.114,322.737,-102.818,173.677,35.080,156.548
C01476=1061.108,322.489,-102.784,173.673,35.075,156.547
C01477=1061.101,322.242,-102.750,173.670,35.071,156.546
C01478=1061.095,321.994,-102.716,173.667,35.066,156.545
C01479=1061.088,321.747,-102.682,173.663,35.062,156.544
C01480=1061.081,321.499,-102.648,173.660,35.058,156.544
C01481=1061.075,321.251,-102.615,173.657,35.053,156.543
C01482=1061.069,321.003,-102.581,173.653,35.049,156.542
C01483=1061.063,320.756,-102.547,173.649,35.044,156.541
C01484=1061.056,320.508,-102.513,173.646,35.040,156.540
C01485=1061.050,320.260,-102.480,173.642,35.036,156.539
C01486=1061.043,320.013,-102.446,173.639,35.031,156.538
C01487=1061.037,319.765,-102.412,173.636,35.027,156.537
C01488=1061.030,319.518,-102.378,173.632,35.022,156.536
C01489=1061.024,319.270,-102.345,173.629,35.018,156.535
C01490=1061.017,319.024,-102.311,173.626,35.013,156.534
C01491=1061.011,318.779,-102.278,173.622,35.009,156.533
C01492=1061.005,318.534,-102.244,173.619,35.005,156.532
C01493=1060.999,318.289,-102.211,173.616,35.001,156.531
C01494=1060.992,318.044,-102.177,173.612,34.996,156.531
C01495=1060.986,317.798,-102.145,173.609,34.992,156.530
C01496=1060.980,317.553,-102.111,173.606,34.988,156.529
C01497=1060.974,317.308,-102.078,173.602,34.983,156.528
C01498=1060.967,317.060,-102.045,173.599,34.979,156.527
C01499=1060.962,316.812,-102.011,173.596,34.974,156.526
C01500=1060.955,316.565,-101.978,173.592,34.970,156.525
C01501=1060.948,316.317,-101.944,173.589,34.966,156.524
C01502=1060.942,316.069,-101.911,173.585,34.961,156.523
C01503=1060.936,315.822,-101.878,173.581,34.957,156.522
C01504=1060.930,315.574,-101.844,173.578,34.953,156.521
C01505=1060.923,315.327,-101.810,173.575,34.948,156.520
C01506=1060.918,315.079,-101.777,173.571,34.944,156.520
C01507=1060.911,314.832,-101.744,173.568,34.940,156.519
C01508=1060.905,314.583,-101.710,173.565,34.935,156.518
C01509=1060.899,314.336,-101.677,173.562,34.931,156.517
C01510=1060.892,314.089,-101.644,173.558,34.926,156.516
C01511=1060.886,313.841,-101.610,173.555,34.922,156.515
C01512=1060.879,313.592,-101.577,173.552,34.918,156.514
C01513=1060.873,313.345,-101.544,173.548,34.914,156.513
C01514=1060.867,313.098,-101.511,173.545,34.909,156.512
C01515=1060.860,312.849,-101.478,173.542,34.905,156.512
C01516=1060.853,312.602,-101.445,173.538,34.901,156.511
C01517=1060.847,312.354,-101.412,173.535,34.897,156.510
C01518=1060.840,312.106,-101.379,173.532,34.893,156.509
C01519=1060.834,311.858,-101.347,173.528,34.889,156.508
C01520=1060.828,311.611,-101.314,173.525,34.885,156.507
C01521=1060.821,311.363,-101.281,173.522,34.881,156.506
C01522=1060.814,311.116,-101.247,173.519,34.877,156.506
C01523=1060.807,310.868,-101.215,173.515,34.872,156.505
C01524=1060.801,310.621,-101.182,173.512,34.868,156.504
C01525=1060.794,310.373,-101.150,173.509,34.864,156.503
C01526=1060.788,310.125,-101.117,173.505,34.860,156.502
C01527=1060.781,309.877,-101.084,173.502,34.855,156.501
C01528=1060.775,309.630,-101.051,173.499,34.851,156.500
C01529=1060.769,309.382,-101.018,173.496,34.847,156.499
C01530=1060.762,309.134,-100.985,173.492,34.843,156.499
C01531=1060.756,308.885,-100.953,173.489,34.839,156.498
C01532=1060.750,308.638,-100.920,173.486,34.835,156.497
C01533=1060.743,308.391,-100.888,173.482,34.831,156.496
C01534=1060.736,308.143,-100.856,173.479,34.827,156.495
C01535=1060.730,307.895,-100.823,173.476,34.823,156.494
C01536=1060.723,307.647,-100.790,173.474,34.818,156.493
C01537=1060.717,307.400,-100.757,173.470,34.814,156.493
C01538=1060.710,307.152,-100.724,173.467,34.810,156.492
C01539=1060.704,306.904,-100.692,173.464,34.806,156.491
C01540=1060.698,306.656,-100.659,173.460,34.802,156.490
C01541=1060.691,306.409,-100.627,173.457,34.798,156.489
C01542=1060.685,306.161,-100.595,173.454,34.794,156.488
C01543=1060.679,305.914,-100.562,173.451,34.790,156.488
C01544=1060.673,305.665,-100.530,173.447,34.785,156.487
C01545=1060.666,305.418,-100.497,173.444,34.781,156.486
C01546=1060.660,305.174,-100.465,173.441,34.777,156.485
C01547=1060.653,304.931,-100.433,173.437,34.773,156.484
C01548=1060.647,304.688,-100.402,173.435,34.769,156.483
C01549=1060.641,304.444,-100.369,173.432,34.765,156.482
C01550=1060.635,304.200,-100.337,173.429,34.761,156.482
C01551=1060.629,303.958,-100.306,173.425,34.757,156.481
C01552=1060.622,303.714,-100.274,173.422,34.753,156.480
C01553=1060.616,303.471,-100.242,173.419,34.749,156.479
C01554=1060.610,303.223,-100.210,173.416,34.745,156.478
C01555=1060.604,302.975,-100.178,173.413,34.741,156.477
C01556=1060.598,302.728,-100.145,173.410,34.737,156.477
C01557=1060.591,302.480,-100.113,173.407,34.732,156.476
C01558=1060.585,302.232,-100.081,173.404,34.728,156.475
C01559=1060.579,301.984,-100.049,173.400,34.724,156.474
C01560=1060.572,301.736,-100.016,173.397,34.720,156.473
C01561=1060.566,301.488,-99.984,173.394,34.716,156.472
C01562=1060.559,301.241,-99.952,173.391,34.712,156.472
C01563=1060.553,300.993,-99.920,173.388,34.708,156.471
C01564=1060.548,300.745,-99.888,173.385,34.704,156.470
C01565=1060.542,300.498,-99.855,173.382,34.699,156.469
C01566=1060.536,300.249,-99.823,173.378,34.695,156.468
C01567=1060.529,300.002,-99.791,173.375,34.691,156.467
C01568=1060.523,299.754,-99.759,173.372,34.687,156.466
C01569=1060.517,299.506,-99.727,173.370,34.683,156.466
C01570=1060.510,299.258,-99.694,173.366,34.679,156.465
C01571=1060.504,299.010,-99.663,173.363,34.675,156.464
C01572=1060.498,298.763,-99.631,173.360,34.671,156.463
C01573=1060.492,298.515,-99.599,173.357,34.667,156.462
C01574=1060.486,298.267,-99.567,173.354,34.663,156.461
C01575=1060.479,298.019,-99.535,173.351,34.659,156.461
C01576=1060.473,297.771,-99.502,173.348,34.655,156.460
C01577=1060.467,297.524,-99.471,173.345,34.650,156.459
C01578=1060.461,297.276,-99.439,173.341,34.646,156.458
C01579=1060.455,297.028,-99.407,173.339,34.642,156.457
C01580=1060.449,296.780,-99.375,173.336,34.638,156.456
C01581=1060.442,296.532,-99.343,173.333,34.634,156.456
C01582=1060.436,296.285,-99.311,173.329,34.630,156.455
C01583=1060.430,296.037,-99.280,173.326,34.626,156.454
C01584=1060.424,295.789,-99.248,173.324,34.622,156.453
C01585=1060.417,295.541,-99.217,173.321,34.618,156.452
C01586=1060.411,295.293,-99.184,173.317,34.614,156.452
C01587=1060.404,295.045,-99.153,173.314,34.610,156.451
C01588=1060.399,294.797,-99.121,173.311,34.606,156.450
C01589=1060.392,294.549,-99.090,173.309,34.602,156.449
C01590=1060.385,294.301,-99.059,173.305,34.598,156.448
C01591=1060.379,294.053,-99.027,173.302,34.594,156.448
C01592=1060.373,293.805,-98.995,173.299,34.591,156.447
C01593=1060.367,293.558,-98.964,173.297,34.586,156.446
C01594=1060.361,293.310,-98.932,173.293,34.582,156.445
C01595=1060.354,293.062,-98.901,173.290,34.579,156.444
C01596=1060.347,292.814,-98.869,173.287,34.575,156.444
C01597=1060.342,292.566,-98.837,173.285,34.570,156.443
C01598=1060.335,292.318,-98.807,173.282,34.567,156.442
C01599=1060.329,292.070,-98.775,173.278,34.563,156.441
C01600=1060.323,291.822,-98.743,173.275,34.559,156.440
C01601=1060.316,291.575,-98.712,173.273,34.555,156.440
C01602=1060.310,291.338,-98.682,173.270,34.551,156.439
C01603=1060.304,291.103,-98.653,173.266,34.547,156.438
C01604=1060.298,290.868,-98.623,173.264,34.544,156.437
C01605=1060.293,290.632,-98.593,173.261,34.540,156.436
C01606=1060.287,290.395,-98.563,173.259,34.536,156.436
C01607=1060.280,290.160,-98.534,173.256,34.532,156.435
C01608=1060.274,289.925,-98.503,173.252,34.528,156.434
C01609=1060.269,289.689,-98.474,173.250,34.525,156.433
C01610=1060.262,289.440,-98.443,173.247,34.521,156.433
C01611=1060.256,289.193,-98.412,173.244,34.517,156.432
C01612=1060.250,288.945,-98.381,173.241,34.513,156.431
C01613=1060.243,288.697,-98.350,173.238,34.509,156.430
C01614=1060.238,288.449,-98.318,173.235,34.505,156.429
C01615=1060.231,288.201,-98.287,173.233,34.502,156.429
C01616=1060.225,287.953,-98.256,173.230,34.497,156.428
C01617=1060.218,287.705,-98.225,173.226,34.493,156.427
C01618=1060.212,287.457,-98.194,173.223,34.490,156.426
C01619=1060.205,287.209,-98.163,173.221,34.485,156.426
C01620=1060.199,286.961,-98.132,173.218,34.482,156.425
C01621=1060.193,286.714,-98.101,173.215,34.478,156.424
C01622=1060.186,286.465,-98.070,173.212,34.474,156.423
C01623=1060.180,286.218,-98.039,173.209,34.470,156.422
C01624=1060.174,285.969,-98.009,173.206,34.466,156.422
C01625=1060.167,285.721,-97.977,173.204,34.462,156.421
C01626=1060.161,285.474,-97.947,173.201,34.459,156.420
C01627=1060.155,285.226,-97.915,173.197,34.454,156.419
C01628=1060.149,284.978,-97.885,173.195,34.451,156.419
C01629=1060.142,284.729,-97.854,173.192,34.447,156.418
C01630=1060.136,284.481,-97.823,173.189,34.443,156.417
C01631=1060.130,284.234,-97.793,173.186,34.439,156.416
C01632=1060.123,283.985,-97.762,173.183,34.435,156.415
C01633=1060.117,283.738,-97.731,173.180,34.431,156.415
C01634=1060.111,283.489,-97.700,173.178,34.428,156.414
C01635=1060.105,283.242,-97.670,173.175,34.423,156.413
C01636=1060.098,282.994,-97.638,173.171,34.420,156.412
C01637=1060.093,282.746,-97.608,173.169,34.416,156.412
C01638=1060.086,282.497,-97.577,173.166,34.412,156.411
C01639=1060.080,282.250,-97.547,173.163,34.408,156.410
C01640=1060.074,282.002,-97.515,173.161,34.404,156.409
C01641=1060.068,281.754,-97.485,173.157,34.400,156.408
C01642=1060.061,281.505,-97.454,173.155,34.397,156.408
C01643=1060.056,281.257,-97.424,173.152,34.392,156.407
C01644=1060.049,281.010,-97.393,173.149,34.389,156.406
C01645=1060.043,280.762,-97.362,173.147,34.385,156.405
C01646=1060.037,280.513,-97.331,173.143,34.381,156.405
C01647=1060.031,280.265,-97.301,173.141,34.377,156.404
C01648=1060.025,280.018,-97.271,173.138,34.373,156.403
C01649=1060.019,279.769,-97.240,173.135,34.369,156.402
C01650=1060.012,279.522,-97.210,173.133,34.366,156.402
C01651=1060.006,279.273,-97.180,173.129,34.361,156.401
C01652=1060.000,279.025,-97.149,173.127,34.358,156.400
C01653=1059.993,278.777,-97.118,173.124,34.354,156.399
C01654=1059.987,278.529,-97.088,173.121,34.350,156.398
C01655=1059.980,278.281,-97.058,173.119,34.346,156.398
C01656=1059.974,278.033,-97.028,173.116,34.342,156.397
C01657=1059.968,277.784,-96.997,173.113,34.339,156.396
C01658=1059.962,277.555,-96.969,173.110,34.335,156.395
C01659=1059.956,277.324,-96.941,173.108,34.331,156.395
C01660=1059.950,277.094,-96.912,173.105,34.328,156.394
C01661=1059.945,276.864,-96.885,173.103,34.324,156.393
C01662=1059.940,276.633,-96.856,173.100,34.321,156.393
C01663=1059.933,276.403,-96.828,173.097,34.317,156.392
C01664=1059.928,276.173,-96.800,173.095,34.314,156.391
C01665=1059.922,275.942,-96.772,173.092,34.310,156.390
C01666=1059.915,275.694,-96.742,173.090,34.306,156.390
C01667=1059.909,275.446,-96.712,173.087,34.302,156.389
C01668=1059.903,275.198,-96.682,173.084,34.299,156.388
C01669=1059.897,274.950,-96.651,173.081,34.295,156.388
C01670=1059.890,274.702,-96.622,173.079,34.291,156.387
C01671=1059.885,274.454,-96.592,173.076,34.287,156.386
C01672=1059.878,274.205,-96.561,173.074,34.284,156.385
C01673=1059.872,273.958,-96.531,173.070,34.279,156.384
C01674=1059.866,273.709,-96.501,173.067,34.276,156.384
C01675=1059.860,273.461,-96.471,173.065,34.272,156.383
C01676=1059.853,273.213,-96.441,173.062,34.268,156.382
C01677=1059.848,272.965,-96.411,173.060,34.264,156.381
C01678=1059.841,272.717,-96.381,173.057,34.260,156.381
C01679=1059.835,272.469,-96.351,173.054,34.257,156.380
C01680=1059.828,272.221,-96.322,173.051,34.253,156.379
C01681=1059.822,271.972,-96.291,173.049,34.249,156.378
C01682=1059.816,271.724,-96.261,173.046,34.245,156.378
C01683=1059.810,271.476,-96.232,173.044,34.242,156.377
C01684=1059.803,271.229,-96.202,173.041,34.237,156.376
C01685=1059.797,270.980,-96.172,173.038,34.234,156.375
C01686=1059.791,270.732,-96.142,173.035,34.230,156.375
C01687=1059.785,270.484,-96.113,173.033,34.226,156.374
C01688=1059.778,270.236,-96.082,173.030,34.222,156.373
C01689=1059.772,269.988,-96.052,173.028,34.219,156.372
C01690=1059.766,269.740,-96.023,173.025,34.215,156.372
C01691=1059.760,269.492,-95.993,173.022,34.211,156.371
C01692=1059.753,269.243,-95.963,173.019,34.207,156.370
C01693=1059.748,268.994,-95.934,173.017,34.203,156.369
C01694=1059.741,268.747,-95.904,173.014,34.200,156.369
C01695=1059.736,268.499,-95.874,173.012,34.196,156.368
C01696=1059.729,268.251,-95.844,173.008,34.192,156.367
C01697=1059.722,268.002,-95.815,173.006,34.188,156.366
C01698=1059.717,267.754,-95.785,173.003,34.185,156.366
C01699=1059.710,267.506,-95.756,173.001,34.180,156.365
C01700=1059.704,267.258,-95.727,172.998,34.177,156.364
C01701=1059.698,267.010,-95.696,172.996,34.173,156.363
C01702=1059.691,266.761,-95.667,172.993,34.170,156.363
C01703=1059.685,266.513,-95.638,172.990,34.165,156.362
C01704=1059.680,266.265,-95.608,172.988,34.162,156.361
C01705=1059.673,266.017,-95.578,172.985,34.158,156.361
C01706=1059.667,265.769,-95.549,172.983,34.154,156.360
C01707=1059.660,265.520,-95.520,172.980,34.150,156.359
C01708=1059.654,265.272,-95.490,172.978,34.147,156.358
C01709=1059.648,265.024,-95.461,172.974,34.143,156.357
C01710=1059.642,264.776,-95.432,172.972,34.139,156.357
C01711=1059.636,264.528,-95.402,172.969,34.135,156.356
C01712=1059.630,264.280,-95.373,172.967,34.132,156.355
C01713=1059.623,264.032,-95.343,172.965,34.128,156.354
C01714=1059.618,263.803,-95.317,172.962,34.124,156.354
C01715=1059.612,263.575,-95.289,172.959,34.121,156.353
C01716=1059.606,263.347,-95.262,172.957,34.117,156.352
C01717=1059.600,263.118,-95.235,172.955,34.114,156.352
C01718=1059.595,262.889,-95.208,172.952,34.110,156.351
C01719=1059.588,262.661,-95.182,172.950,34.107,156.350
C01720=1059.583,262.432,-95.155,172.948,34.103,156.350
C01721=1059.577,262.204,-95.128,172.946,34.100,156.349
C01722=1059.571,261.956,-95.099,172.942,34.096,156.348
C01723=1059.564,261.708,-95.070,172.940,34.093,156.348
C01724=1059.558,261.460,-95.041,172.937,34.089,156.347
C01725=1059.552,261.211,-95.012,172.935,34.085,156.346
C01726=1059.546,260.963,-94.983,172.932,34.082,156.346
C01727=1059.539,260.715,-94.954,172.930,34.078,156.345
C01728=1059.533,260.466,-94.924,172.928,34.074,156.344
C01729=1059.526,260.218,-94.895,172.924,34.070,156.343
C01730=1059.520,259.970,-94.866,172.922,34.067,156.343
C01731=1059.513,259.722,-94.838,172.919,34.063,156.342
C01732=1059.507,259.474,-94.809,172.917,34.059,156.341
C01733=1059.501,259.225,-94.780,172.915,34.056,156.340
C01734=1059.495,258.977,-94.751,172.912,34.052,156.340
C01735=1059.488,258.729,-94.722,172.910,34.048,156.339
C01736=1059.482,258.481,-94.693,172.906,34.044,156.338
C01737=1059.476,258.233,-94.664,172.904,34.041,156.338
C01738=1059.470,257.985,-94.635,172.902,34.037,156.337
C01739=1059.464,257.736,-94.607,172.899,34.033,156.336
C01740=1059.457,257.488,-94.578,172.897,34.029,156.335
C01741=1059.451,257.239,-94.548,172.895,34.026,156.335
C01742=1059.444,256.991,-94.519,172.892,34.022,156.334
C01743=1059.438,256.743,-94.490,172.889,34.018,156.333
C01744=1059.431,256.494,-94.463,172.886,34.014,156.332
C01745=1059.425,256.246,-94.434,172.884,34.010,156.332
C01746=1059.419,255.998,-94.405,172.882,34.007,156.331
C01747=1059.413,255.749,-94.376,172.879,34.003,156.330
C01748=1059.407,255.502,-94.348,172.877,34.000,156.330
C01749=1059.401,255.254,-94.318,172.875,33.995,156.329
C01750=1059.395,255.005,-94.290,172.872,33.992,156.328
C01751=1059.389,254.757,-94.261,172.869,33.988,156.327
C01752=1059.383,254.509,-94.232,172.867,33.985,156.327
C01753=1059.376,254.260,-94.204,172.864,33.980,156.326
C01754=1059.370,254.012,-94.175,172.862,33.977,156.325
C01755=1059.363,253.764,-94.146,172.860,33.973,156.324
C01756=1059.358,253.515,-94.118,172.857,33.969,156.324
C01757=1059.351,253.267,-94.089,172.855,33.965,156.323
C01758=1059.345,253.018,-94.061,172.852,33.962,156.322
C01759=1059.339,252.770,-94.032,172.849,33.958,156.321
C01760=1059.332,252.522,-94.004,172.847,33.954,156.321
C01761=1059.326,252.274,-93.975,172.845,33.950,156.320
C01762=1059.321,252.026,-93.947,172.842,33.946,156.319
C01763=1059.315,251.777,-93.918,172.840,33.943,156.319
C01764=1059.309,251.529,-93.889,172.838,33.939,156.318
C01765=1059.302,251.281,-93.860,172.835,33.935,156.317
C01766=1059.296,251.032,-93.832,172.832,33.931,156.316
C01767=1059.289,250.784,-93.804,172.830,33.928,156.316
C01768=1059.283,250.535,-93.775,172.828,33.924,156.315
C01769=1059.278,250.288,-93.747,172.825,33.920,156.314
C01770=1059.272,250.058,-93.720,172.823,33.916,156.313
C01771=1059.267,249.829,-93.694,172.821,33.913,156.313
C01772=1059.261,249.599,-93.668,172.819,33.910,156.312
C01773=1059.255,249.369,-93.641,172.817,33.906,156.311
C01774=1059.250,249.140,-93.615,172.814,33.902,156.311
C01775=1059.244,248.911,-93.589,172.812,33.899,156.310
C01776=1059.238,248.682,-93.563,172.810,33.895,156.309
C01777=1059.232,248.452,-93.537,172.808,33.892,156.309
C01778=1059.227,248.204,-93.509,172.805,33.888,156.308
C01779=1059.221,247.956,-93.480,172.803,33.884,156.307
C01780=1059.215,247.707,-93.451,172.801,33.881,156.306
C01781=1059.208,247.458,-93.424,172.799,33.876,156.306
C01782=1059.203,247.211,-93.395,172.795,33.873,156.305
C01783=1059.197,246.962,-93.367,172.793,33.869,156.304
C01784=1059.191,246.713,-93.338,172.791,33.865,156.303
C01785=1059.185,246.465,-93.310,172.789,33.861,156.303
C01786=1059.178,246.218,-93.282,172.786,33.858,156.302
C01787=1059.172,245.969,-93.254,172.784,33.853,156.301
C01788=1059.166,245.720,-93.226,172.782,33.850,156.301
